		gst_datensatz.st_wkz.nockenschaltwerk_bestueckachse.arr_nocken[NO_BW_BANDFAENGER_EINFAHREN].b_camvalid := FALSE;
		gst_datensatz.st_wkz.nockenschaltwerk_bestueckachse.arr_nocken[NO_BW_BANDFAENGER_AUSFAHREN].b_camvalid := FALSE;
		gst_datensatz.st_wkz.nockenschaltwerk_bestueckachse.arr_nocken[NO_BW_BANDKLEMMEN_EINFAHREN].b_camvalid := FALSE;
		gst_datensatz.st_wkz.nockenschaltwerk_bestueckachse.arr_nocken[NO_BW_BANDKLEMMEN_AUSFAHREN].b_camvalid := FALSE;
		gst_datensatz.st_wkz.nockenschaltwerk_bestueckachse.arr_nocken[NO_UW_BANDFAENGER_EINFAHREN].b_camvalid := FALSE;
		gst_datensatz.st_wkz.nockenschaltwerk_bestueckachse.arr_nocken[NO_UW_BANDFAENGER_AUSFAHREN].b_camvalid := FALSE;
		gst_datensatz.st_wkz.nockenschaltwerk_bestueckachse.arr_nocken[NO_UW_BANDKLEMMEN_EINFAHREN].b_camvalid := FALSE;
		gst_datensatz.st_wkz.nockenschaltwerk_bestueckachse.arr_nocken[NO_UW_BANDKLEMMEN_AUSFAHREN].b_camvalid := FALSE;

		gst_datensatz.st_wkz.nockenschaltwerk_bestueckachse.arr_nocken[NO_PNEUMATIKBANDEINZUG_GLS].b_camvalid := FALSE;
		gst_datensatz.st_wkz.nockenschaltwerk_bestueckachse.arr_nocken[NO_UW_BESTUECKSCHIEBER_ON].b_camvalid := FALSE;
		gst_datensatz.st_wkz.nockenschaltwerk_bestueckachse.arr_nocken[NO_UW_BESTUECKSCHIEBER_OFF].b_camvalid := FALSE;
		gst_datensatz.st_wkz.nockenschaltwerk_bestueckachse.arr_nocken[SP_UW_BESTUECKSCHIEBER_ON].b_camvalid := FALSE;
		gst_datensatz.st_wkz.nockenschaltwerk_bestueckachse.arr_nocken[SP_UW_BESTUECKSCHIEBER_OFF].b_camvalid := FALSE;


		zyl_bandfaenger.fb.b_no_gesteuert_im_norm_betrieb := TRUE;
		zyl_bandklemmen.fb.b_no_gesteuert_im_norm_betrieb := TRUE;

		zyl_bandfaenger.fb.b_no_gesteuert_im_norm_betrieb := TRUE;
		zyl_bandklemmen.fb.b_no_gesteuert_im_norm_betrieb := TRUE;

END_CASE;
END_ACTION
ACTION subr_ST_Bandeinzugsnocken_ein:
CASE gst_datensatz.st_wkz.i16_typ_bandeinzug OF
	 STANDARD_2FACH_V2:

		(* Bandeinzug: Standard_2fach_V2 *)
		gst_datensatz.st_wkz.nockenschaltwerk_bestueckachse.arr_nocken[NO_BW_BANDFAENGER_LI_EINFAHREN].b_camvalid := TRUE;
		gst_datensatz.st_wkz.nockenschaltwerk_bestueckachse.arr_nocken[NO_BW_BANDFAENGER_LI_AUSFAHREN].b_camvalid := TRUE;
		gst_datensatz.st_wkz.nockenschaltwerk_bestueckachse.arr_nocken[NO_BW_BANDKLEMMEN_LI_EINFAHREN].b_camvalid := TRUE;
		gst_datensatz.st_wkz.nockenschaltwerk_bestueckachse.arr_nocken[NO_BW_BANDKLEMMEN_LI_AUSFAHREN].b_camvalid := TRUE;
		gst_datensatz.st_wkz.nockenschaltwerk_bestueckachse.arr_nocken[NO_UW_BANDFAENGER_LI_EINFAHREN].b_camvalid := TRUE;
		gst_datensatz.st_wkz.nockenschaltwerk_bestueckachse.arr_nocken[NO_UW_BANDFAENGER_LI_AUSFAHREN].b_camvalid := TRUE;
		gst_datensatz.st_wkz.nockenschaltwerk_bestueckachse.arr_nocken[NO_UW_BANDKLEMMEN_LI_EINFAHREN].b_camvalid := TRUE;
		gst_datensatz.st_wkz.nockenschaltwerk_bestueckachse.arr_nocken[NO_UW_BANDKLEMMEN_LI_AUSFAHREN].b_camvalid := TRUE;
		gst_datensatz.st_wkz.nockenschaltwerk_bestueckachse.arr_nocken[NO_BW_BANDFAENGER_RE_EINFAHREN].b_camvalid := TRUE;
		gst_datensatz.st_wkz.nockenschaltwerk_bestueckachse.arr_nocken[NO_BW_BANDFAENGER_RE_AUSFAHREN].b_camvalid := TRUE;
		gst_datensatz.st_wkz.nockenschaltwerk_bestueckachse.arr_nocken[NO_BW_BANDKLEMMEN_RE_EINFAHREN].b_camvalid := TRUE;
		gst_datensatz.st_wkz.nockenschaltwerk_bestueckachse.arr_nocken[NO_BW_BANDKLEMMEN_RE_AUSFAHREN].b_camvalid := TRUE;
		gst_datensatz.st_wkz.nockenschaltwerk_bestueckachse.arr_nocken[NO_UW_BANDFAENGER_RE_EINFAHREN].b_camvalid := TRUE;
		gst_datensatz.st_wkz.nockenschaltwerk_bestueckachse.arr_nocken[NO_UW_BANDFAENGER_RE_AUSFAHREN].b_camvalid := TRUE;
		gst_datensatz.st_wkz.nockenschaltwerk_bestueckachse.arr_nocken[NO_UW_BANDKLEMMEN_RE_EINFAHREN].b_camvalid := TRUE;
		gst_datensatz.st_wkz.nockenschaltwerk_bestueckachse.arr_nocken[NO_UW_BANDKLEMMEN_RE_AUSFAHREN].b_camvalid := TRUE;
		(* Bandeinzug: Standard_2fach_V2 *)
		gst_datensatz.st_wkz.nockenschaltwerk_bestueckachse.arr_nocken[NO_BW_BANDFAENGER_LI_BAEZV2_EINFAHREN].b_camvalid := TRUE;
		gst_datensatz.st_wkz.nockenschaltwerk_bestueckachse.arr_nocken[NO_BW_BANDFAENGER_LI_BAEZV2_AUSFAHREN].b_camvalid := TRUE;
		gst_datensatz.st_wkz.nockenschaltwerk_bestueckachse.arr_nocken[NO_BW_BANDKLEMMEN_LI_BAEZV2_EINFAHREN].b_camvalid := TRUE;
		gst_datensatz.st_wkz.nockenschaltwerk_bestueckachse.arr_nocken[NO_BW_BANDKLEMMEN_LI_BAEZV2_AUSFAHREN].b_camvalid := TRUE;
		gst_datensatz.st_wkz.nockenschaltwerk_bestueckachse.arr_nocken[NO_BW_BANDFAENGER_RE_BAEZV2_EINFAHREN].b_camvalid := TRUE;
		gst_datensatz.st_wkz.nockenschaltwerk_bestueckachse.arr_nocken[NO_BW_BANDFAENGER_RE_BAEZV2_AUSFAHREN].b_camvalid := TRUE;
		gst_datensatz.st_wkz.nockenschaltwerk_bestueckachse.arr_nocken[NO_BW_BANDKLEMMEN_RE_BAEZV2_EINFAHREN].b_camvalid := TRUE;
		gst_datensatz.st_wkz.nockenschaltwerk_bestueckachse.arr_nocken[NO_BW_BANDKLEMMEN_RE_BAEZV2_AUSFAHREN].b_camvalid := TRUE;

		zyl_bandfaenger_li.fb.b_no_gesteuert_im_norm_betrieb := FALSE;
		zyl_bandklemmen_li.fb.b_no_gesteuert_im_norm_betrieb := FALSE;
		zyl_bandfaenger_re.fb.b_no_gesteuert_im_norm_betrieb := FALSE;
		zyl_bandklemmen_re.fb.b_no_gesteuert_im_norm_betrieb := FALSE;

	BANDWECHSLER_V2:
		(* Klemmbandeinzug ohne Sensoren *)
		gst_datensatz.st_wkz.nockenschaltwerk_bestueckachse.arr_nocken[NO_BW_BANDFAENGER_BAWEV2_EINFAHREN].b_camvalid := TRUE;
		gst_datensatz.st_wkz.nockenschaltwerk_bestueckachse.arr_nocken[NO_BW_BANDFAENGER_BAWEV2_AUSFAHREN].b_camvalid := TRUE;
		gst_datensatz.st_wkz.nockenschaltwerk_bestueckachse.arr_nocken[NO_BW_BANDKLEMMEN_BAWEV2_EINFAHREN].b_camvalid := TRUE;
		gst_datensatz.st_wkz.nockenschaltwerk_bestueckachse.arr_nocken[NO_BW_BANDKLEMMEN_BAWEV2_AUSFAHREN].b_camvalid := TRUE;

		gst_datensatz.st_wkz.nockenschaltwerk_bestueckachse.arr_nocken[NO_BW_BANDFAENGER_EINFAHREN].b_camvalid := TRUE;
		gst_datensatz.st_wkz.nockenschaltwerk_bestueckachse.arr_nocken[NO_BW_BANDFAENGER_AUSFAHREN].b_camvalid := TRUE;
		gst_datensatz.st_wkz.nockenschaltwerk_bestueckachse.arr_nocken[NO_BW_BANDKLEMMEN_EINFAHREN].b_camvalid := TRUE;
		gst_datensatz.st_wkz.nockenschaltwerk_bestueckachse.arr_nocken[NO_BW_BANDKLEMMEN_AUSFAHREN].b_camvalid := TRUE;
		gst_datensatz.st_wkz.nockenschaltwerk_bestueckachse.arr_nocken[NO_UW_BANDFAENGER_EINFAHREN].b_camvalid := TRUE;
		gst_datensatz.st_wkz.nockenschaltwerk_bestueckachse.arr_nocken[NO_UW_BANDFAENGER_AUSFAHREN].b_camvalid := TRUE;
		gst_datensatz.st_wkz.nockenschaltwerk_bestueckachse.arr_nocken[NO_UW_BANDKLEMMEN_EINFAHREN].b_camvalid := TRUE;
		gst_datensatz.st_wkz.nockenschaltwerk_bestueckachse.arr_nocken[NO_UW_BANDKLEMMEN_AUSFAHREN].b_camvalid := TRUE;

		gst_datensatz.st_wkz.nockenschaltwerk_bestueckachse.arr_nocken[NO_PNEUMATIKBANDEINZUG_GLS].b_camvalid := TRUE;
		gst_datensatz.st_wkz.nockenschaltwerk_bestueckachse.arr_nocken[NO_UW_BESTUECKSCHIEBER_ON].b_camvalid := b_bestueckschieber_ueberwachung_aktiv;
		gst_datensatz.st_wkz.nockenschaltwerk_bestueckachse.arr_nocken[NO_UW_BESTUECKSCHIEBER_OFF].b_camvalid := b_bestueckschieber_ueberwachung_aktiv;
		gst_datensatz.st_wkz.nockenschaltwerk_bestueckachse.arr_nocken[SP_UW_BESTUECKSCHIEBER_ON].b_camvalid := b_bestueckschieber_ueberwachung_aktiv;
		gst_datensatz.st_wkz.nockenschaltwerk_bestueckachse.arr_nocken[SP_UW_BESTUECKSCHIEBER_OFF].b_camvalid := b_bestueckschieber_ueberwachung_aktiv;

		zyl_bandfaenger.fb.b_no_gesteuert_im_norm_betrieb := TRUE;
		zyl_bandklemmen.fb.b_no_gesteuert_im_norm_betrieb := TRUE;
END_CASE;
END_ACTION
ACTION subr_ST_Bandeinzugsnocken_li_ein:
CASE gst_datensatz.st_wkz.i16_typ_bandeinzug OF
	STANDARD_2FACH_V2:

		(* Bandeinzug: Standard_2fach_V1 *)
		gst_datensatz.st_wkz.nockenschaltwerk_bestueckachse.arr_nocken[NO_BW_BANDFAENGER_LI_EINFAHREN].b_camvalid := TRUE;
		gst_datensatz.st_wkz.nockenschaltwerk_bestueckachse.arr_nocken[NO_BW_BANDFAENGER_LI_AUSFAHREN].b_camvalid := TRUE;
		gst_datensatz.st_wkz.nockenschaltwerk_bestueckachse.arr_nocken[NO_BW_BANDKLEMMEN_LI_EINFAHREN].b_camvalid := TRUE;
		gst_datensatz.st_wkz.nockenschaltwerk_bestueckachse.arr_nocken[NO_BW_BANDKLEMMEN_LI_AUSFAHREN].b_camvalid := TRUE;
		gst_datensatz.st_wkz.nockenschaltwerk_bestueckachse.arr_nocken[NO_UW_BANDFAENGER_LI_EINFAHREN].b_camvalid := TRUE;
		gst_datensatz.st_wkz.nockenschaltwerk_bestueckachse.arr_nocken[NO_UW_BANDFAENGER_LI_AUSFAHREN].b_camvalid := TRUE;
		gst_datensatz.st_wkz.nockenschaltwerk_bestueckachse.arr_nocken[NO_UW_BANDKLEMMEN_LI_EINFAHREN].b_camvalid := TRUE;
		gst_datensatz.st_wkz.nockenschaltwerk_bestueckachse.arr_nocken[NO_UW_BANDKLEMMEN_LI_AUSFAHREN].b_camvalid := TRUE;
		(* Bandeinzug: Standard_2fach_V2 *)
		gst_datensatz.st_wkz.nockenschaltwerk_bestueckachse.arr_nocken[NO_BW_BANDFAENGER_LI_BAEZV2_EINFAHREN].b_camvalid := TRUE;
		gst_datensatz.st_wkz.nockenschaltwerk_bestueckachse.arr_nocken[NO_BW_BANDFAENGER_LI_BAEZV2_AUSFAHREN].b_camvalid := TRUE;
		gst_datensatz.st_wkz.nockenschaltwerk_bestueckachse.arr_nocken[NO_BW_BANDKLEMMEN_LI_BAEZV2_EINFAHREN].b_camvalid := TRUE;
		gst_datensatz.st_wkz.nockenschaltwerk_bestueckachse.arr_nocken[NO_BW_BANDKLEMMEN_LI_BAEZV2_AUSFAHREN].b_camvalid := TRUE;

		zyl_bandfaenger_li.fb.b_no_gesteuert_im_norm_betrieb := FALSE;
		zyl_bandklemmen_li.fb.b_no_gesteuert_im_norm_betrieb := FALSE;
		zyl_bandfaenger_re.fb.b_no_gesteuert_im_norm_betrieb := FALSE;
		zyl_bandklemmen_re.fb.b_no_gesteuert_im_norm_betrieb := FALSE;

END_CASE;
END_ACTION
ACTION subr_ST_Bandeinzugsnocken_re_ein:
CASE gst_datensatz.st_wkz.i16_typ_bandeinzug OF
	STANDARD_2FACH_V2:

		(* Bandeinzug: Standard_2fach_V1 *)
		gst_datensatz.st_wkz.nockenschaltwerk_bestueckachse.arr_nocken[NO_BW_BANDFAENGER_RE_EINFAHREN].b_camvalid := TRUE;
		gst_datensatz.st_wkz.nockenschaltwerk_bestueckachse.arr_nocken[NO_BW_BANDFAENGER_RE_AUSFAHREN].b_camvalid := TRUE;
		gst_datensatz.st_wkz.nockenschaltwerk_bestueckachse.arr_nocken[NO_BW_BANDKLEMMEN_RE_EINFAHREN].b_camvalid := TRUE;
		gst_datensatz.st_wkz.nockenschaltwerk_bestueckachse.arr_nocken[NO_BW_BANDKLEMMEN_RE_AUSFAHREN].b_camvalid := TRUE;
		gst_datensatz.st_wkz.nockenschaltwerk_bestueckachse.arr_nocken[NO_UW_BANDFAENGER_RE_EINFAHREN].b_camvalid := TRUE;
		gst_datensatz.st_wkz.nockenschaltwerk_bestueckachse.arr_nocken[NO_UW_BANDFAENGER_RE_AUSFAHREN].b_camvalid := TRUE;
		gst_datensatz.st_wkz.nockenschaltwerk_bestueckachse.arr_nocken[NO_UW_BANDKLEMMEN_RE_EINFAHREN].b_camvalid := TRUE;
		gst_datensatz.st_wkz.nockenschaltwerk_bestueckachse.arr_nocken[NO_UW_BANDKLEMMEN_RE_AUSFAHREN].b_camvalid := TRUE;
		(* Bandeinzug: Standard_2fach_V2 *)
		gst_datensatz.st_wkz.nockenschaltwerk_bestueckachse.arr_nocken[NO_BW_BANDFAENGER_RE_BAEZV2_EINFAHREN].b_camvalid := TRUE;
		gst_datensatz.st_wkz.nockenschaltwerk_bestueckachse.arr_nocken[NO_BW_BANDFAENGER_RE_BAEZV2_AUSFAHREN].b_camvalid := TRUE;
		gst_datensatz.st_wkz.nockenschaltwerk_bestueckachse.arr_nocken[NO_BW_BANDKLEMMEN_RE_BAEZV2_EINFAHREN].b_camvalid := TRUE;
		gst_datensatz.st_wkz.nockenschaltwerk_bestueckachse.arr_nocken[NO_BW_BANDKLEMMEN_RE_BAEZV2_AUSFAHREN].b_camvalid := TRUE;
		
		zyl_bandfaenger_li.fb.b_no_gesteuert_im_norm_betrieb := FALSE;
		zyl_bandklemmen_li.fb.b_no_gesteuert_im_norm_betrieb := FALSE;
		zyl_bandfaenger_re.fb.b_no_gesteuert_im_norm_betrieb := FALSE;
		zyl_bandklemmen_re.fb.b_no_gesteuert_im_norm_betrieb := FALSE;

END_CASE;
END_ACTION
ACTION subr_ST_Cam_B_Achse:
(* B-Achse *)
fb_axis_b_achse.st_camscaling_data.SlaveScaling :=
	F_Servobandeinzug_Strecke_zu_Grad(
		strecke := INT_TO_LREAL(gst_datensatz.st_bestueckprogramm.i16_b[i16_bestueckposzaehler])
			* gst_datensatz.st_band.r_raster);

IF b_achse.Status.CamScalingPending THEN
	st_sm.b_skalierung_noch_aktiv := TRUE;
	fb_state_entry.i16_next_step := FEHLER;
ELSE
	IF b_achse.NcToPlc.CoupleState = 0 THEN
		st_drive_cmd_b_achse.enu_cmd := CAM_IN_SLAVE;
	ELSE
		st_drive_cmd_b_achse.enu_cmd := CAM_SCALEING_SLAVE;
	END_IF
END_IF
END_ACTION
ACTION subr_ST_Cam_Bestueck_Maschine:
CASE gst_datensatz.st_md.i16_typ_zelle OF
	KEINE_ZELLE:
		;
	BESTUECKZELLE_1700, BESTUECKZELLE_1720:
		subr_ST_Cam_Bestueckachse();

	RASTERFOLIE:
		;
END_CASE
END_ACTION
ACTION subr_ST_Cam_Bestueckachse:
(* Bestueckachse *)
IF gst_datensatz.st_bestueckprogramm.i16_b[i16_bestueckposzaehler] <= 0 THEN
	i16_bestueckachse_cam_table_id := 6;	(* 0-Scalierung *)
	subr_ST_Bandeinzugsnocken_aus();
ELSE
	i16_bestueckachse_cam_table_id := 5;	(* 1-Scalierung *)
	subr_ST_Bandeinzugsnocken_ein();
END_IF

IF i16_bestueckachse_cam_table_id <> i16_bestueckachse_cam_table_id_alt THEN
	fb_axis_bestueckachse.mc_activation_mode_camin:= MC_CAMACTIVATION_ATMASTERCAMPOS;
	fb_axis_bestueckachse.lr_activation_position_camin := gst_datensatz.st_md.st_md_bestueckachse.lr_startposition;
	st_drive_cmd_bestueckachse.enu_cmd := CAM_IN_SLAVE;
	i16_bestueckachse_cam_table_id_alt := i16_bestueckachse_cam_table_id;
END_IF
END_ACTION
ACTION subr_ST_Cam_Y_Achse:
(* Y-Achse *)
IF i16_bestueckposzaehler = 0 THEN
	lr_ErsteBestueckposY := gst_datensatz.st_isk.lr_pos_y_0 +
						gst_datensatz.st_wkz.lr_offset_y_pos_0 +
						gst_datensatz.st_wt.lr_offset_y_pos_0 +
						gst_datensatz.st_md.lr_offset_y_pos_0 +
						gst_datensatz.st_bestueckprogramm.lr_y[0];
	fb_axis_y_achse.st_camscaling_data.SlaveScaling := fb_berechnung_override_achse.lr_skalierung_slave_achse2 := lr_ErsteBestueckposY - y_achse.NcToPlc.ActPos;
	(* Falls die Positionierung Probleme macht, könnte man auch so rechnen *)
	(*fb_axis_y_achse.st_camscaling_data.SlaveScaling := fb_berechnung_override_achse.lr_skalierung_slave_achse2 := lr_ErsteBestueckposY - gst_datensatz.st_wkz.r_wkz_einfahrpos_y;*)
ELSIF i16_bestueckposzaehler > 0 AND i16_bestueckposzaehler < gst_datensatz.st_bestueckprogramm.i32_anzahl THEN
	fb_axis_y_achse.st_camscaling_data.SlaveScaling := fb_berechnung_override_achse.lr_skalierung_slave_achse2 := gst_datensatz.st_bestueckprogramm.lr_y[i16_bestueckposzaehler] - gst_datensatz.st_bestueckprogramm.lr_y[i16_bestueckposzaehler - 1];
ELSE
	fb_axis_y_achse.st_camscaling_data.SlaveScaling := fb_berechnung_override_achse.lr_skalierung_slave_achse2 := 0.0;
END_IF
IF y_achse.Status.CamScalingPending THEN
	st_sm.b_skalierung_noch_aktiv := TRUE;
	fb_state_entry.i16_next_step := FEHLER;
ELSE
	IF y_achse.NcToPlc.CoupleState = 0 THEN
		st_drive_cmd_y_achse.enu_cmd := CAM_IN_SLAVE;
	ELSE
		st_drive_cmd_y_achse.enu_cmd := CAM_SCALEING_SLAVE;
	END_IF
END_IF
END_ACTION
ACTION subr_ST_Cam_Z_Achse:
(* Z-Achse *)
IF i16_bestueckposzaehler > 0 AND i16_bestueckposzaehler < gst_datensatz.st_bestueckprogramm.i32_anzahl THEN
	fb_axis_z_achse.st_camscaling_data.SlaveScaling := fb_berechnung_override_achse.lr_skalierung_slave_achse1 := gst_datensatz.st_bestueckprogramm.lr_z[i16_bestueckposzaehler] - gst_datensatz.st_bestueckprogramm.lr_z[i16_bestueckposzaehler - 1];
ELSE
	fb_axis_z_achse.st_camscaling_data.SlaveScaling := fb_berechnung_override_achse.lr_skalierung_slave_achse1 := 0.0;
END_IF
IF z_achse.Status.CamScalingPending THEN
	st_sm.b_skalierung_noch_aktiv := TRUE;
	fb_state_entry.i16_next_step := FEHLER;
ELSE
	IF z_achse.NcToPlc.CoupleState = 0 THEN
		st_drive_cmd_z_achse.enu_cmd := CAM_IN_SLAVE;
	ELSE
		st_drive_cmd_z_achse.enu_cmd := CAM_SCALEING_SLAVE;
	END_IF
END_IF
END_ACTION
ACTION subr_ST_EinzugLueften:
(* SP_SERVOBANDEINZUG_LUEFTEN niemals vorsteuern *)
gst_datensatz.st_wkz.nockenschaltwerk_bestueckachse.arr_nocken[SP_SERVOBANDEINZUG_LUEFTEN].t_vorsteuerzeit := t#0ms;

fb_r_trig_bandeinzug_lueften(CLK:= nockenschaltwerk_bestueckachse.fb.arr_spur[SP_SERVOBANDEINZUG_LUEFTEN], Q=> );
fb_f_trig_bandeinzug_lueften(CLK:= nockenschaltwerk_bestueckachse.fb.arr_spur[SP_SERVOBANDEINZUG_LUEFTEN], Q=> );

(* Abschalten, falls die Schrittkette beim Lüften aus irgendwelchen Gründen hängen bleibt *)
IF fb_r_trig_bandeinzug_lueften.Q AND
	i16_step_lueften > 0 THEN
		sm_fehler_achse_lueften := TRUE;
		fb_state_entry.i16_next_step := FEHLER;
END_IF


(* Schrittkette zum Einzug in Regelung setzen mit Positionsangleich  *)
CASE i16_step_lueften OF
(*=======================================================*)
	0:	(* CAM Out bei R Trig Lueftnocke *)

		(*-----------------------Weiterschaltbedingungen----------------------------*)
		IF fb_r_trig_bandeinzug_lueften.Q AND
			bestueckachse.NcToPlc.CoupleState <> 0 AND
			((NOT b_einfaedeln_aktiv_servo AND
			(* Bei einer Umfahrung soll Servo nicht lüften, weil die Fänger des WKZ das Band nicht halten *)
			gst_datensatz.st_bestueckprogramm.i16_b[i16_bestueckposzaehler] >= 1 ) OR
			(b_einfaedeln_aktiv_servo AND
			i16_einfaedelzaehler >= gst_datensatz.st_wkz.i16_einfaedelhub_lueften)) THEN		(* Nach x Einfädelhüben ist Band sicher im WKZ, dann darf Servobaneinzug wieder entlüften *)
			st_drive_cmd_b_achse.enu_cmd := CAM_OUT_SLAVE;
			i16_step_lueften := 10;
		END_IF

(*=======================================================*)
	10:

		(*-----------------------Weiterschaltbedingungen----------------------------*)
		IF st_drive_cmd_b_achse.enu_cmd = NO_COMMAND THEN
			ST_Servobandeinzug.i_Stromlimit := ST_Servobandeinzug.i16_lueft_torque;
			i16_step_lueften := 20;
		END_IF

(*=======================================================*)
	20: (* HOME Servobandeinzug bei F Trig Lueftnocke *)

		(*-----------------------Weiterschaltbedingungen----------------------------*)
		IF fb_f_trig_bandeinzug_lueften.Q THEN
			axis_bandeinzug_achse.st_ctrl.in.b_home := TRUE;
			i16_step_lueften := 30;
		END_IF

(*=======================================================*)
	30:

		(*-----------------------Weiterschaltbedingungen----------------------------*)
		IF axis_bandeinzug_achse.st_ctrl.out.b_fertig_2 THEN
			axis_bandeinzug_achse.st_ctrl.in.b_home := FALSE;
			i16_step_lueften := 0;
		END_IF

END_CASE
END_ACTION
ACTION subr_ST_PosUW_Bestueckachse:
(* Wenn die Betückachse von der Virtuellen Achse entkoppelt wird, muss dauerhaft der OT Sensor belegt sein.
Überwachung, ob das Auskoppeln rechtzeitig gemacht wird. Ab 300 Hub gibt es Probleme *)
IF i16_bestueckachse_cam_table_id = 6 AND NOT ST_Bestueckachse.e_referenz_sensor THEN
	sm_fehler_positionierung_bestueckachse := TRUE;
	fb_state_entry.i16_next_step := FEHLER;
END_IF
END_ACTION
ACTION subr_ST_PosUW_YZ_Achse:
(* Y *)
(* Kontrolle der Skalierungsposition der Achse nach dem Setzen eines Pins *)
IF ABS(y_achse.NcToPlc.ActPos - (lr_merker_y_pos + gst_datensatz.st_bestueckprogramm.lr_y[i16_bestueckposzaehler])) > 0.1THEN
	sm_fehler_bestueckposition_y := TRUE;
	fb_state_entry.i16_next_step := FEHLER;
END_IF

(* Überwachung auf Kommando abgeschlossen. Zusätzliche Kontrolle auf Ausführung des Skalierungskommandos *)
IF st_drive_cmd_y_achse.enu_cmd <> NO_COMMAND THEN
	st_sm.b_ende_camming_nocke := TRUE;
	fb_state_entry.i16_next_step := FEHLER;
END_IF

(* Z *)
(* Kontrolle der Skalierungsposition der Achse nach dem Setzen eines Pins *)
IF ABS(z_achse.NcToPlc.ActPos - (lr_merker_z_pos + gst_datensatz.st_bestueckprogramm.lr_z[i16_bestueckposzaehler])) > 0.2THEN
	sm_fehler_bestueckposition_z := TRUE;
	fb_state_entry.i16_next_step := FEHLER;
END_IF

(* Überwachung auf Kommando abgeschlossen. Zusätzliche Kontrolle auf Ausführung des Skalierungskommandos *)
IF st_drive_cmd_z_achse.enu_cmd <> NO_COMMAND THEN
	st_sm.b_ende_camming_nocke := TRUE;
	fb_state_entry.i16_next_step := FEHLER;
END_IF

(* Pythagoras YZ *)
(*	tv + gg: 10.08.2021
	Wir müssen nicht nur jede Achse einzeln überwachen, sondern beide Achsen zusammen überwachen.
	Bsp. 74pol 2-Fach WT: Es gibt hier Sprünge die nur 0.04 in Y Verschoben, welche dann die 
	Überwachung in Y-Achse ausgelöst hat, obwohl alles funktionert hat. Z Pos ist um 5 mm verschoben*)

(* Kontrolle, ob die Achsen gegenüber dem letzten Bestückhub weiter gefahren ist *)
lr_merker_y_pos_neu := y_achse.NcToPlc.ActPos;
lr_merker_z_pos_neu := z_achse.NcToPlc.ActPos;

lr_abstand_yz := SQRT(	EXPT(lr_merker_y_pos_alt - lr_merker_y_pos_neu, 2) +
						EXPT(lr_merker_z_pos_alt - lr_merker_z_pos_neu, 2));

IF 	(fb_axis_y_achse.st_camscaling_data.SlaveScaling <> 0 OR
	fb_axis_z_achse.st_camscaling_data.SlaveScaling <> 0) AND
	lr_abstand_yz < 0.05
THEN
	sm_fehler_positionierung_y := TRUE;
	sm_fehler_positionierung_z := TRUE;
	fb_state_entry.i16_next_step := FEHLER;
END_IF

lr_merker_y_pos_alt := lr_merker_y_pos_neu;
lr_merker_z_pos_alt := lr_merker_z_pos_neu;
END_ACTION
ACTION subr_ST_PosUW_Z_Achse:
(* Kontrolle der Skalierungsposition der Achse nach dem Setzen eines Pins *)
IF ABS(z_achse.NcToPlc.ActPos - (lr_merker_z_pos + gst_datensatz.st_bestueckprogramm.lr_z[i16_bestueckposzaehler])) > 0.2THEN
	sm_fehler_bestueckposition_z := TRUE;
	fb_state_entry.i16_next_step := FEHLER;
END_IF

(* Überwachung auf Kommando abgeschlossen. Zusätzliche Kontrolle auf Ausführung des Skalierungskommandos *)
IF st_drive_cmd_z_achse.enu_cmd <> NO_COMMAND THEN
	st_sm.b_ende_camming_nocke := TRUE;
	fb_state_entry.i16_next_step := FEHLER;
END_IF

(* Kontrolle, ob die Achse gegenüber dem letzten Bestückhub weiter gefahren ist *)
lr_merker_z_pos_neu := z_achse.NcToPlc.ActPos;
IF fb_axis_z_achse.st_camscaling_data.SlaveScaling <> 0 THEN
	IF ABS(lr_merker_z_pos_alt - lr_merker_z_pos_neu) > 0.05 THEN
		lr_merker_z_pos_alt := lr_merker_z_pos_neu;
	ELSE
		sm_fehler_positionierung_z := TRUE;
		fb_state_entry.i16_next_step := FEHLER;
	END_IF
END_IF
END_ACTION

(* POU EPT Lib/Funktionsbausteine/ST_BerechnungOverride, ST *)
FUNCTION_BLOCK ST_BerechnungOverride
VAR_INPUT
	i16_betriebsart				: enum_betriebsarten;
	lr_skalierung_slave_achse1		: LREAL;
	lr_skalierung_slave_achse2		: LREAL;
	lr_override_vorgabe			: LREAL;
	lr_faktor						: LREAL;

	lr_FaktorHub				: LREAL;
	lr_HubAuto					: LREAL;
END_VAR
VAR_OUTPUT
	lr_override					: LREAL := 0.0;
END_VAR
VAR
	lr_offset						: LREAL := 100.0;
	tmp_lr_override_slave1		: LREAL := 0.0;
	tmp_lr_override_slave2		: LREAL := 0.0;

	lr_ProzentDerRichtdrehzahl	: LREAL;
	lr_Reduzierung				: LREAL;
END_VAR
(* Funktion zur Berechnung des Override der  Masterachse: y = - faktor * x^2 + offset *)
(* Die Funktion besteht aus einer auf dem Kopf stehenden Parabel, welche um den faktor nach oben verschoben ist *)
(* Aufpassen bei den Nullstellen der Funktion, wenn faktor und offset verändert werden *)

(* Die Anpassung der maximalen Mastergeschwindigkeit an die Verfahrlänge des Slaves wird hier einfach über eine empirisch ermittelte Funktion realisiert *)
(* Eine verbesserte Anpassung stellt die Berechnung der maximalen Mastergeschwindigkeit (ST_MFMaxMasterVelo) im CamEditor dar. *)

tmp_lr_override_slave1 := - lr_faktor * (lr_skalierung_slave_achse1 * lr_skalierung_slave_achse1)  + lr_offset;
tmp_lr_override_slave2 := - lr_faktor * (lr_skalierung_slave_achse2 * lr_skalierung_slave_achse2)  + lr_offset;

IF tmp_lr_override_slave1 < 0.0 THEN
	 tmp_lr_override_slave1 := 0.0;
ELSIF tmp_lr_override_slave1 >= 100.0 THEN
	 tmp_lr_override_slave1 := 100.0;
END_IF
IF tmp_lr_override_slave2 < 0.0 THEN
	 tmp_lr_override_slave2 := 0.0;
ELSIF tmp_lr_override_slave2 >= 100.0 THEN
	 tmp_lr_override_slave2 := 100.0;
END_IF

IF i16_betriebsart = AUTO THEN
	(* Nur wenn der mit der Funktion berechnete Override kleiner ist, als die Vorgabe, dann wird der Funktionswert übernommen *)
	IF 	tmp_lr_override_slave1 < lr_override_vorgabe OR
		tmp_lr_override_slave2 < lr_override_vorgabe THEN

		IF tmp_lr_override_slave1 <= tmp_lr_override_slave2 THEN
			lr_override := tmp_lr_override_slave1;
		ELSIF tmp_lr_override_slave2 < tmp_lr_override_slave1 THEN
			lr_override := tmp_lr_override_slave2;
		ELSE
			lr_override := lr_override_vorgabe;
		END_IF

	ELSE
		lr_override := lr_override_vorgabe;
	END_IF
ELSE
	lr_override := lr_override_vorgabe;
END_IF


(*neue Berechnung==========================================================================*)
(*Reduzierung abhängig von der Nenndrehzahl*)
lr_ProzentDerRichtdrehzahl:=(lr_HubAuto *100)/250;
IF	lr_HubAuto >250 AND
	lr_override_vorgabe > lr_override THEN
	lr_override := 100-((lr_override_vorgabe - lr_override) * (lr_ProzentDerRichtdrehzahl /100)) ;
END_IF

(*nur Reduzieren wenn das Ergebniss kleiner ist als bei der Reduzierung durch die Pin Anzahl*)
lr_Reduzierung:= (lr_override_vorgabe - lr_override)/100;
IF	(1 - lr_Reduzierung) < lr_FaktorHub THEN
	lr_override := lr_override;
ELSE
	lr_override:= 100 * lr_FaktorHub;
END_IF

IF	lr_override > lr_override_vorgabe OR
	lr_override < 0 THEN
	lr_override:= lr_override_vorgabe;
END_IF

(*Beim Einfädeln wird der Override vom Bausstein ST_TippTasten einfach durchgeschleust*)
IF	ST_TippTasten.b_einfaedeln_aktiv OR
	ST_TippTasten.b_initialisierungsphase THEN
	lr_override := lr_override_vorgabe;
END_IF

(*bei Prüfteilen Override fest auf 30% *)
IF	lr_override_vorgabe > 30 AND
	(FIND( gst_datensatz.st_md.s_aktuelle_artikelnummer,'ruef') <> 0 OR FIND( gst_datensatz.st_md.s_aktuelle_artikelnummer,'erth') <> 0)THEN
	lr_override := 30;
END_IF
END_FUNCTION_BLOCK

(* POU Gemeinsamkeiten17xx/Achsen/ST_Servobandeinzug, ST *)
PROGRAM ST_Servobandeinzug
VAR_INPUT
	st_config_achse						: struct_ecd_config;
	st_ctrl_in								: struct_ctrl_in;
	e_steuerung_ein						: BOOL;
	e_ba_mit_bedingungen				: BOOL;
	e_tuere_vorne_offen					: BOOL;
	e_tuere_hinten_offen					: BOOL;
	i_Stromlimit							: INT;		(* Werte zwischen 0 und 1000 möglich*)
END_VAR
VAR_IN_OUT
	st_visu								: struct_ecd_visu;
END_VAR
VAR_OUTPUT
	st_ctrl_out							: struct_ctrl_out;
END_VAR
VAR
	st_sm						 		: struct_ecd_meldungen;
	st_drive_cmd							: struct_ecd_cmd;
	fb_ton_wz							: TON;
	fb_ton_quitt							: TON;
	fb_r_trig_taste_plus					: R_TRIG;
	fb_r_trig_taste_minus					: R_TRIG;
	fb_r_trig_bremse						: R_TRIG;
	fb_r_trig_tippen						: R_TRIG;
	fb_r_trig_hand_dialog					: R_TRIG;
	fb_axis								: ST_AxisJobCtrl_Motion;
	fb_state_entry							: ST_StateEntry;
	fb_ton_uez							: TON;
	b_ibn_start							: BOOL := FALSE;
	fb_r_trig_ibn_start						: R_TRIG;
	fb_ton_ibn_start						: TON;
	fb_ton_wz_rueckzug					: TON;
	fb_tof_gls_ref							: TOF;
	fb_r_trig_gls_ref						: R_TRIG;
	fb_ton_wz_disable						: TON;
	fb_ton_wz_param						: TON;
	i									: UINT := 0;
	fb_r_trig_limit_sensor_positiv			: R_TRIG;
	fb_r_trig_limit_sensor_negativ			: R_TRIG;
	fb_r_trig_achse_lueften					: R_TRIG;
	b_referenzieren						: BOOL := FALSE;

	b_hand_dialog_aktiv					: BOOL := FALSE;
	st_geschwindigkeiten					: struct_ecd_geschwindigkeiten;
	i_zaehler_steigende_flanke				: INT;	(* Zähler für Bandvorschubkontrolle Gabellichtschranke *)
	i_zaehler_fallende_flanke				: INT;	(* Zähler für Bandvorschubkontrolle Gabellichtschranke *)
	fb_r_trig_vorschubkontrolle				: R_TRIG;
	fb_f_trig_vorschubkontrolle				: F_TRIG;
	fb_r_trig_nocke_einzug					: R_TRIG;
	fb_f_trig_nocke_einzug					: F_TRIG;
	i16_max_torque						: INT := 1000;
	i16_lueft_torque						: INT := 2;	(* sehr klein, damit sich Band ausrichten kann und Servo nicht dagegen arbeitet *)
	i16_man_einfaedel_torque				: INT := 30;
	i16_auto_einfaedel_torque				: INT := 150;
	i16_einfaedel_torque					: INT := 20;
	i16_block_torque						: INT := 40;
	lr_rueckzugposition					: LREAL := 0.5;
	b_merker_bremse						: BOOL := FALSE;
	b_merker_bremse_auf_zu				: BOOL := FALSE;
	r_raster_alt							: REAL := 0.0;
	i16_raster_nc_parameter				: INT := 0;
	b_merker_lueften						: BOOL := FALSE;
	b_merker_regeln						: BOOL := FALSE;

	err_id								: DWORD := 0;

	mc_set_cam_online_change_mode		: MC_SetCamOnlineChangeMode;

	lr_posmerker_an_faenger				: LREAL := 0;

	sm_bandrueckzug						: BOOL := FALSE;
	sm_bandreferenzieren					: BOOL := FALSE;
	sm_fehler_bandvorschub				: BOOL := FALSE;
	sm_fehler_raster						: BOOL := FALSE;
	sm_fehler_bandeinfaedeln				: BOOL := FALSE;
	sm_fahren_auf_gls					: BOOL := FALSE;
	sm_band_rausgezogen				: BOOL := FALSE;
	sm_band_nicht_in_lichtschranke			: BOOL := FALSE;

	e_limit_sensor_positive				AT %I* : BOOL;
	e_limit_sensor_negative				AT %I* : BOOL;
	e_gls_bandreferenzieren				AT %I* : BOOL;	(* Sensor dient auch als Vorschubkontrolle *)
	i16_torque							AT %I* : INT;
	i16_vorgabe_stromlimit					AT %Q* : INT;

	i16_debug 							: INT;

	(* Lueften *)
	fb_r_trig_bandeinzug_lueften			: R_TRIG;

	lr_merker_pos_vor_lueften				: LREAL := 0.0;
	lr_merker_pos_nach_lueften			: LREAL := 0.0;
	lr_merker_pos_diff_lueften				: LREAL := 0.0;

	lr_startpos							: LREAL := 0;

END_VAR

VAR CONSTANT
	lr_konst_strecke_ls_bandeinzug			: LREAL := 70;
	lr_max_strecke_gls_wkz				: LREAL := 110;
END_VAR
(* Zeiten *)
fb_ton_wz(IN:= , PT:= , Q=>  , ET=> );
fb_ton_uez(IN:= , PT:= , Q=>  , ET=> );
fb_ton_wz_rueckzug(IN:= , PT:= t#300ms, Q=> , ET=> );
fb_tof_gls_ref(IN:= e_gls_bandreferenzieren, PT:= t#150ms, Q=>  , ET=> );
fb_ton_wz_disable(IN:= , PT:= t#500ms, Q=> , ET=> );
fb_ton_wz_param(IN:= , PT:= t#500ms, Q=> , ET=> );
fb_ton_quitt(IN:= , PT:= t#100ms, Q=> , ET=> );


(* Flanken *)
fb_r_trig_limit_sensor_positiv(CLK:= st_config_achse.b_limitsensor_positiv_vorhanden AND NOT e_limit_sensor_positive, Q=> );
fb_r_trig_limit_sensor_negativ(CLK:= st_config_achse.b_limitsensor_negativ_vorhanden AND NOT e_limit_sensor_negative, Q=> );
fb_r_trig_taste_plus(CLK:= ST_Euchner_Handbedienpult.b_Taste_Plus, Q=> );
fb_r_trig_taste_minus(CLK:= ST_Euchner_Handbedienpult.b_Taste_Minus, Q=> );
fb_r_trig_bremse(CLK:= visu_hinten.out.ST_Servobandeinzug.b_taste_bremse, Q=> );
fb_r_trig_tippen(CLK:= visu_hinten.out.ST_Servobandeinzug.b_taste_tippen, Q=> );
fb_r_trig_gls_ref(CLK:= e_gls_bandreferenzieren, Q=> );
fb_r_trig_vorschubkontrolle(CLK:= e_gls_bandreferenzieren, Q=> );
fb_f_trig_vorschubkontrolle(CLK:= e_gls_bandreferenzieren, Q=> );

fb_r_trig_hand_dialog(CLK:= b_hand_dialog_aktiv, Q=> );

fb_f_trig_nocke_einzug(CLK:= nockenschaltwerk_bestueckachse.fb.arr_spur[SP_SERVOBANDEINZUG_GLS], Q=> );
fb_r_trig_nocke_einzug(CLK:= nockenschaltwerk_bestueckachse.fb.arr_spur[SP_SERVOBANDEINZUG_GLS], Q=> );

(* Inbetriebnahme *)
fb_r_trig_ibn_start (CLK:= b_ibn_start , Q=> );
fb_ton_ibn_start (IN:= , PT:= t#1s, Q=> , ET=> );

i16_debug := fb_state_entry.i16_step;

IF fb_r_trig_ibn_start .Q THEN
	fb_ton_ibn_start .IN := TRUE;
ELSE
	IF fb_ton_ibn_start .Q THEN
		b_ibn_start  := FALSE;
	 	fb_ton_ibn_start .IN := FALSE;
	END_IF
END_IF

(* Vorgabewert an Regler übergeben*)
i16_vorgabe_stromlimit := i_Stromlimit;

(* Achse steuern *)
IF fb_state_entry.i16_step >= 500 AND fb_state_entry.i16_step < 700 THEN
	fb_axis.lr_override_vorgabe := 3.0;
ELSIF fb_state_entry.i16_step >= 700 AND fb_state_entry.i16_step < 800 THEN
	fb_axis.lr_override_vorgabe := 25.0;
ELSE
	fb_axis.lr_override_vorgabe := ST_TippTasten.lr_override;
END_IF

fb_axis(
	e_referenznocken:= ,
	b_refsensor_vorhanden:= st_config_achse.b_refsensor_vorhanden,
	b_limitsensor_positiv_vorhanden:= st_config_achse.b_limitsensor_positiv_vorhanden,
	b_limitsensor_negativ_vorhanden:= st_config_achse.b_limitsensor_negativ_vorhanden,
	i16_achstyp := st_config_achse.i16_achstyp,
	st_position:= ,
	lr_override_vorgabe:= ,
	mc_richtung_modulo:= ,
	mc_richtung_velocity:= ,
	mc_referenzmodus:= ,
	mc_buffermode_axis:= ,
	ui16_soeparam_write_value:= ,
	w_idn:= ,
	i16_nc_parameter_nummer:= ,
	r_wert_nc_write_parameter:= ,
	st_vorgabe_geschwindigkeiten:= st_geschwindigkeiten,
	lr_soll_geschwindigkeit:=,
	b_bedingung_sls:= NOT e_tuere_vorne_offen OR NOT e_tuere_hinten_offen,
	st_ads_info := ,
	st_eccoe_sdo := ,
	st_masterachse:= b_achse,
	st_visu_axis:= st_visu,
	st_ecd_cmd:= st_drive_cmd,
	ui16_soeparam_read_value=> ,
	r_wert_nc_read_parameter=> );

(* Achse mit dem Euchner Handbediengerät vorwärts und rückwärts Bewegen*)
IF ST_Betriebsarten.i16_betriebsart = HAND AND fb_r_trig_hand_dialog.Q THEN
	fb_state_entry.i16_next_step := HANDRAD;
END_IF

(* Visualisierung des Bremsenzustandes am Backpanel *)
IF fb_axis.ui16_soeparam_write_value = 0 THEN
	 visu_hinten.in.b_zustand_bremse := FALSE;
ELSIF fb_axis.ui16_soeparam_write_value = 2 THEN
	 visu_hinten.in.b_zustand_bremse := TRUE;
END_IF

(* Motorbremse von Hand am Backpanel öffnen *)
IF fb_r_trig_bremse.Q THEN
	fb_ton_wz_disable.IN := FALSE;
	fb_ton_wz_param.IN := FALSE;
	b_merker_bremse := TRUE;
END_IF

IF b_merker_bremse THEN
	(* Reglerfreigabe wegnehmen/setzen und Motorbremse auf/zu *)
	IF NOT fb_ton_wz_disable.IN AND NOT fb_ton_wz_param.IN THEN
		IF b_merker_bremse_auf_zu THEN
			(* Bremse ZU *)
			st_drive_cmd.enu_cmd := POWER_ENABLE;
			fb_axis.ui16_soeparam_write_value := 0;
			b_merker_bremse_auf_zu := FALSE;
		ELSE
			(* Bremse AUF *)
			st_drive_cmd.enu_cmd := POWER_DISABLE;
			fb_axis.ui16_soeparam_write_value := 2;
			b_merker_bremse_auf_zu := TRUE;
		END_IF
		fb_ton_wz_disable.IN := TRUE;
	END_IF

	IF fb_ton_wz_disable.Q AND st_drive_cmd.enu_cmd = NO_COMMAND THEN
		fb_axis.w_idn := P_0_IDN + 96;
		st_drive_cmd.enu_cmd := SOE_WRITE_PARAM;
		fb_ton_wz_disable.IN := FALSE;
		fb_ton_wz_param.IN := TRUE;
	END_IF

	IF fb_ton_wz_param.Q AND st_drive_cmd.enu_cmd = NO_COMMAND THEN
		fb_ton_wz_param.IN := FALSE;
		b_merker_bremse := FALSE;
	END_IF
END_IF

(* Vorschubkontrolle des Bandes *)
IF fb_state_entry.i16_next_step >= BEREIT AND fb_state_entry.i16_next_step < 400 THEN
	subr_ST_Vorschubkontrolle();
END_IF

(* =======================================Toplevel========================================== *)
(* Starte Inbetriebnahme-Sequenz *)
IF st_ctrl_in.b_gehe_step_ibn THEN
	fb_state_entry.i16_next_step := INBETRIEBNAHME;
END_IF

IF (NOT e_steuerung_ein OR NOT e_ba_mit_bedingungen) AND y_achse.Status.Operational THEN
	st_drive_cmd.enu_cmd := POWER_DISABLE;
END_IF

IF fb_state_entry.i16_next_step > INIT AND fb_state_entry.i16_next_step < FEHLER THEN
	(* =====Fehler vom Achskontroller===== *)
	IF st_drive_cmd.b_job_fehler THEN
		fb_state_entry.i16_next_step := FEHLER;
	END_IF

	IF fb_state_entry.i16_next_step > 70 THEN
		(* Devicefehler *)
		IF b_achse.Status.Error THEN
			st_sm.b_achsfehler := TRUE;
			(*  Bei einem Achsfehler des Servomotors wird das Drehmoment weggeschalten, um ein Zerstören des Igelrads zu vermeiden. *)
			i_Stromlimit := i16_lueft_torque;
			fb_state_entry.i16_next_step := FEHLER;
		ELSIF b_achse.Status.DriveDeviceError THEN
			st_sm.b_devicefehler := TRUE;
			fb_state_entry.i16_next_step := FEHLER;
		END_IF
	END_IF

	IF fb_state_entry.i16_next_step < STOP THEN
		(* =====Achse wird gestoppt===== *)
		IF st_ctrl_in.b_stop THEN
			fb_state_entry.i16_next_step := STOP;
		ELSIF fb_state_entry.i16_next_step < HALT THEN
			(* =====Achse wird angehalten===== *)
			IF st_ctrl_in.b_halt THEN
				fb_state_entry.i16_next_step := HALT;
			END_IF
		END_IF
	END_IF
END_IF

(* ==================================Schrittkette================================ *)
fb_state_entry(
	i16_next_step:= ,
	i16_pos:= 1,
	s_debugtext:= ,
	E=> ,
	X=> ,
	i16_step=> ,
	i16_last_step=> );

CASE fb_state_entry.i16_step OF
(*=======================================================*)
	INIT_OBJ:
		IF st_config_achse.b_config_fertig THEN
			fb_state_entry.i16_next_step := 1;
		END_IF

(*=======================================================*)
	1:	(* Warte bis NetID´s der Slaves ausgelesen sind *)
		IF fb_state_entry.E THEN
			;
		END_IF

		(*-----------------------Weiterschaltbedingungen----------------------------*)
		IF ST_EthercatDiag.st_ctrl_out.b_fertig THEN
			fb_state_entry.i16_next_step := 2;
		END_IF

(*=======================================================*)
	2:	(* Spezifische NC-Achsparameter auslesen *)
		IF fb_state_entry.E THEN
			fb_axis.i16_nc_parameter_nummer := MaxVelocitySystem;
			st_drive_cmd.enu_cmd := READ_NC_PARAMETER;
		END_IF

		(*-----------------------Weiterschaltbedingungen----------------------------*)
		IF st_drive_cmd.enu_cmd = NO_COMMAND THEN
			st_geschwindigkeiten.lr_auto_max := fb_axis.r_wert_nc_read_parameter;
			st_geschwindigkeiten.lr_maximalgeschwindigkeit := fb_axis.r_wert_nc_read_parameter;
			st_geschwindigkeiten.lr_auto_min := 1;
			st_geschwindigkeiten.lr_jog := 50;
			fb_state_entry.i16_next_step := 3;
		END_IF

(*=======================================================*)
	3:	(* Spezifische NC-Achsparameter auslesen *)
		IF fb_state_entry.E THEN
			fb_axis.i16_nc_parameter_nummer := MaxAccelerationSystem;
			st_drive_cmd.enu_cmd := READ_NC_PARAMETER;
		END_IF

		(*-----------------------Weiterschaltbedingungen----------------------------*)
		IF st_drive_cmd.enu_cmd = NO_COMMAND THEN
			st_geschwindigkeiten.lr_beschleunigung := fb_axis.r_wert_nc_read_parameter;
			fb_state_entry.i16_next_step := 4;
		END_IF

(*=======================================================*)
	4:	(* Spezifische NC-Achsparameter auslesen *)
		IF fb_state_entry.E THEN
			fb_axis.i16_nc_parameter_nummer := MaxDecelerationSystem;
			st_drive_cmd.enu_cmd := READ_NC_PARAMETER;
		END_IF

		(*-----------------------Weiterschaltbedingungen----------------------------*)
		IF st_drive_cmd.enu_cmd = NO_COMMAND THEN
			st_geschwindigkeiten.lr_verzoegerung := fb_axis.r_wert_nc_read_parameter;
			fb_state_entry.i16_next_step := 5;
		END_IF

(*=======================================================*)
	5:	(* Spezifische NC-Achsparameter auslesen *)
		IF fb_state_entry.E THEN
			fb_axis.i16_nc_parameter_nummer := MaxJerk;
			st_drive_cmd.enu_cmd := READ_NC_PARAMETER;
		END_IF

		(*-----------------------Weiterschaltbedingungen----------------------------*)
		IF st_drive_cmd.enu_cmd = NO_COMMAND THEN
			st_geschwindigkeiten.lr_ruck := fb_axis.r_wert_nc_read_parameter;
			fb_state_entry.i16_next_step := 6;
		END_IF

(*=======================================================*)
	6:	(* Konfigurationen der Achse *)
		IF fb_state_entry.E THEN
			fb_axis.st_eccoe_sdo.s_ec_slave_net_id := ST_EthercatDiag.s_ec_slave_net_id[2];
			fb_axis.st_eccoe_sdo.ui16_slave_addr := st_config_achse.ui16_ethercat_adr;
		END_IF

		(*-----------------------Weiterschaltbedingungen----------------------------*)
		fb_state_entry.i16_next_step := FEHLER; (*in Fehler gehen damit die Achsen resetet werden. Sonst steigen die Achsen bei einem TC Restart aus*)

(*=======================================================*)
	INIT:
		IF fb_state_entry.E THEN
			fb_ton_wz.IN := FALSE;
			fb_ton_uez.IN	:= FALSE;
			fb_ton_quitt.IN := FALSE;
			fb_ton_wz_rueckzug.IN := FALSE;
			fb_tof_gls_ref.IN := FALSE;
			fb_ton_wz_disable.IN := FALSE;
			b_referenzieren := FALSE;
			sm_bandrueckzug := FALSE;
			sm_bandreferenzieren := FALSE;
			sm_fehler_bandvorschub := FALSE;
			sm_fehler_raster := FALSE;
			sm_fehler_bandeinfaedeln := FALSE;
			sm_fahren_auf_gls := FALSE;
			sm_band_rausgezogen := FALSE;
			sm_band_nicht_in_lichtschranke := FALSE;
			st_sm.b_achse_nicht_auf_startpos := FALSE;
			st_sm.b_achsfehler := FALSE;
			st_sm.b_devicefehler := FALSE;
			st_sm.b_keine_verfahrfreigabe := FALSE;
			st_sm.b_ende_skalierungs_nocke := FALSE;
			st_sm.b_ende_camming_nocke := FALSE;
			st_sm.b_skalierung_noch_aktiv := FALSE;
			st_ctrl_out.b_fehler := FALSE;
			st_ctrl_out.b_fertig := FALSE;
			st_ctrl_out.b_fertig_2 := FALSE;
			st_ctrl_out.b_bereit := FALSE;
			st_ctrl_out.b_prebereit := FALSE;
			st_ctrl_out.b_bandende := FALSE;
			st_ctrl_out.b_bremse_geoeffnet := FALSE;
			st_ctrl_out.b_bremse_geschlossen := FALSE;
			st_ctrl_out.b_servo_auf_einfaedelpos := FALSE;
			i16_max_torque := 1000;
			i16_lueft_torque := 2;	(* sehr klein, damit sich Band ausrichten kann und Servo nicht dagegen arbeitet *)
			i16_man_einfaedel_torque := 30;
			i16_auto_einfaedel_torque := 150;
			i16_einfaedel_torque := 20;
			i16_block_torque := 40;
			i_Stromlimit := i16_max_torque;
			mc_set_cam_online_change_mode.Execute := FALSE;

			fb_axis.lr_soll_geschwindigkeit := gst_datensatz.st_wkz.r_auto_bandeinzug;
		END_IF

		(*-----------------------Weiterschaltbedingungen----------------------------*)
		IF st_ctrl_in.b_preinit THEN
			fb_state_entry.i16_next_step := 20;
		END_IF

(*=======================================================*)
	20:	(* Schleppabstandsüberwachung einschalten *)
		IF fb_state_entry.E THEN
			fb_axis.r_wert_nc_write_parameter := 1;
			fb_axis.i16_nc_parameter_nummer := EnablePosLagMonitoring;
			st_drive_cmd.enu_cmd := WRITE_NC_PARAMETER;
		END_IF

		(*-----------------------Weiterschaltbedingungen----------------------------*)
		IF st_drive_cmd.enu_cmd = NO_COMMAND THEN
			fb_state_entry.i16_next_step := 25;
		END_IF

(*=======================================================*)
	25:	(* Abfrage auf geändertes Raster *)

		(*-----------------------Weiterschaltbedingungen----------------------------*)
		IF r_raster_alt = gst_datensatz.st_band.r_raster THEN
			fb_state_entry.i16_next_step := 60;
		ELSE
			fb_state_entry.i16_next_step := 30;	(* Rasterwechsel -> NC-Parameter müssen neu eingelesen werden! *)
		END_IF

(*=======================================================*)
	30:	(* Konfiguration der Achse in Abhängigkeit des Igelrades/Rasters *)
		(* Die Werte wurden in der Achs-Konfiguration des Systemmanagers für die verschiedenen Raster berechnet *)
		IF fb_state_entry.E THEN
			fb_state_entry.i16_next_step := 41;
		END_IF

(*=======================================================*)
	41:	(* Spezifische NC-Achsparameter auslesen *)
		IF fb_state_entry.E THEN
			fb_axis.i16_nc_parameter_nummer := MaxVelocitySystem;
			st_drive_cmd.enu_cmd := READ_NC_PARAMETER;
		END_IF

		(*-----------------------Weiterschaltbedingungen----------------------------*)
		IF st_drive_cmd.enu_cmd = NO_COMMAND THEN
			st_geschwindigkeiten.lr_auto_max := fb_axis.r_wert_nc_read_parameter;
			st_geschwindigkeiten.lr_maximalgeschwindigkeit := fb_axis.r_wert_nc_read_parameter;
			st_geschwindigkeiten.lr_auto_min := 1;
			st_geschwindigkeiten.lr_jog :=360;
			fb_state_entry.i16_next_step := 42;
		END_IF

(*=======================================================*)
	42:	(* Spezifische NC-Achsparameter auslesen *)
		IF fb_state_entry.E THEN
			fb_axis.i16_nc_parameter_nummer := MaxAccelerationSystem;
			st_drive_cmd.enu_cmd := READ_NC_PARAMETER;
		END_IF

		(*-----------------------Weiterschaltbedingungen----------------------------*)
		IF st_drive_cmd.enu_cmd = NO_COMMAND THEN
			st_geschwindigkeiten.lr_beschleunigung := fb_axis.r_wert_nc_read_parameter;
			fb_state_entry.i16_next_step := 43;
		END_IF

(*=======================================================*)
	43:	(* Spezifische NC-Achsparameter auslesen *)
		IF fb_state_entry.E THEN
			fb_axis.i16_nc_parameter_nummer := MaxDecelerationSystem;
			st_drive_cmd.enu_cmd := READ_NC_PARAMETER;
		END_IF

		(*-----------------------Weiterschaltbedingungen----------------------------*)
		IF st_drive_cmd.enu_cmd = NO_COMMAND THEN
			st_geschwindigkeiten.lr_verzoegerung := fb_axis.r_wert_nc_read_parameter;
			fb_state_entry.i16_next_step := 44;
		END_IF

(*=======================================================*)
	44:	(* Spezifische NC-Achsparameter auslesen *)
		IF fb_state_entry.E THEN
			fb_axis.i16_nc_parameter_nummer := MaxJerk;
			st_drive_cmd.enu_cmd := READ_NC_PARAMETER;
		END_IF

		(*-----------------------Weiterschaltbedingungen----------------------------*)
		IF st_drive_cmd.enu_cmd = NO_COMMAND THEN
			st_geschwindigkeiten.lr_ruck := fb_axis.r_wert_nc_read_parameter;
			fb_state_entry.i16_next_step := 45;
		END_IF

(*=======================================================*)
	45:	(* Bremse auf "automtisch" stellen. *)
		IF fb_state_entry.E THEN
			fb_axis.w_idn := P_0_IDN + 96;
			fb_axis.ui16_soeparam_write_value := 0;
			st_drive_cmd.enu_cmd := SOE_WRITE_PARAM;
		END_IF

		(*-----------------------Weiterschaltbedingungen----------------------------*)
		IF st_drive_cmd.enu_cmd = NO_COMMAND THEN
			fb_state_entry.i16_next_step := 50;
		END_IF

(*=======================================================*)
	50:	(* Änderungen im Camtable mit Eigenschaft: "mit sofortiger Wirkung" aktivieren *)
		IF fb_state_entry.E THEN
			mc_set_cam_online_change_mode.ActivationMode := MC_CAMACTIVATION_INSTANTANEOUS;
			mc_set_cam_online_change_mode.MasterScalingMode := MC_CAMSCALING_USERDEFINED;
			mc_set_cam_online_change_mode.SlaveScalingMode := MC_CAMSCALING_USERDEFINED;
			mc_set_cam_online_change_mode.CamTableID := 4;
			mc_set_cam_online_change_mode.Execute := TRUE;
		END_IF

		(*-----------------------Weiterschaltbedingungen----------------------------*)
		IF mc_set_cam_online_change_mode.Done THEN
			mc_set_cam_online_change_mode.Execute := FALSE;
			fb_state_entry.i16_next_step := 55;
		ELSIF mc_set_cam_online_change_mode.Error THEN
			err_id := mc_set_cam_online_change_mode.ErrorID;
			fb_state_entry.i16_next_step := FEHLER;
		END_IF

(*=======================================================*)
	55:	(* Überprüfe Nullpunktverschiebung des Absolutwertgebers auf Korrektheit *)
		IF fb_state_entry.E THEN
			fb_axis.i16_nc_parameter_nummer := AxisEncoderOffset;	(* vom Datentyp MC_AxisParameter *)
			st_drive_cmd.enu_cmd := READ_NC_PARAMETER;
		END_IF

		(*-----------------------Weiterschaltbedingungen----------------------------*)
		IF st_drive_cmd.enu_cmd = NO_COMMAND THEN
			IF fb_axis.r_wert_nc_read_parameter = gst_datensatz.st_md.st_md_b_achse.lr_nullpunktverschiebung THEN
				fb_state_entry.i16_next_step := 60;	(* Reglerfreigabe setzen *)
			ELSE
				fb_state_entry.i16_next_step := 56;	(* Nullpunktverschiebung schreiben *)
			END_IF
		END_IF

(*=======================================================*)
	56:	(* Nullpunktverschiebung hat sich geändert, deshalb erst Null reinschreiben, um keinen Additionsfehler zu machen, *)
		(* weil der Wert der Verschiebung beim Neustart komplett auf die Achse geschrieben wird *)
		IF fb_state_entry.E THEN
			fb_axis.i16_nc_parameter_nummer := AxisEncoderOffset;
			fb_axis.r_wert_nc_write_parameter := 0.0;
			st_drive_cmd.enu_cmd := WRITE_NC_PARAMETER;
		END_IF

		(*-----------------------Weiterschaltbedingungen----------------------------*)
		IF st_drive_cmd.enu_cmd = NO_COMMAND THEN
			fb_state_entry.i16_next_step := 57;
		END_IF

(*=======================================================*)
	57:	(* Aktuelle Nullpunktverschiebung des Absolutwertgebers an die Achse senden *)
		IF fb_state_entry.E THEN
			fb_axis.i16_nc_parameter_nummer := AxisEncoderOffset;
			fb_axis.r_wert_nc_write_parameter := gst_datensatz.st_md.st_md_b_achse.lr_nullpunktverschiebung;
			st_drive_cmd.enu_cmd := WRITE_NC_PARAMETER;
		END_IF

		(*-----------------------Weiterschaltbedingungen----------------------------*)
		IF st_drive_cmd.enu_cmd = NO_COMMAND THEN
			fb_state_entry.i16_next_step := 60;
		END_IF

(*=======================================================*)
	60:	(* Reglerfreigabe setzen , Reset wird bei Bedarf automatisch ausgeführt*)
		IF fb_state_entry.E THEN
			st_drive_cmd.enu_cmd := POWER_ENABLE;
		END_IF

		(*-----------------------Weiterschaltbedingungen----------------------------*)
		IF st_drive_cmd.enu_cmd = NO_COMMAND THEN
			fb_state_entry.i16_next_step := 70;
		END_IF

(*=======================================================*)
	70:	(* Nullpunktverschiebung ist geschrieben *)
		IF fb_state_entry.E THEN
			st_ctrl_out.b_prebereit := TRUE;
		END_IF

		(*-----------------------Weiterschaltbedingungen----------------------------*)
		IF st_ctrl_in.b_init THEN
			fb_state_entry.i16_next_step := BEREIT;
		END_IF

(*=======================================================*)
	BEREIT:
		IF fb_state_entry.E THEN
			b_referenzieren := FALSE;
			st_ctrl_out.b_bereit := TRUE;
		END_IF

		(*-----------------------Weiterschaltbedingungen----------------------------*)
		IF st_ctrl_in.b_bremse_auf THEN
			fb_state_entry.i16_next_step := 200;	(* Motorbremse lösen *)
		ELSIF st_ctrl_in.b_bremse_zu THEN
			fb_state_entry.i16_next_step := 300;	(* Motorbremse fest *)
		ELSIF st_ctrl_in.b_home THEN
			fb_state_entry.i16_next_step := 400;	(* HOME *)
			st_ctrl_out.b_fertig_2 := FALSE;
		ELSIF st_ctrl_in.b_start THEN
			st_ctrl_out.b_fertig := FALSE;
			st_ctrl_out.b_fertig_2 := FALSE;
			fb_state_entry.i16_next_step := 500;	(* Einfädelprozedur *)
		ELSIF st_ctrl_in.b_ausfaedeln_servo THEN
			fb_state_entry.i16_next_step := 700;	(* Band ausfädeln *)
		ELSIF st_ctrl_in.b_startpos THEN
			st_ctrl_out.b_servo_auf_einfaedelpos := FALSE;
			fb_state_entry.i16_next_step := 800; (*Igelrad auf Startposition fahren*)
		END_IF

(*=======================================================*)
	200:	(* Reglerfreigabe wegnehmen *)
		IF fb_state_entry.E THEN
			st_drive_cmd.enu_cmd := POWER_DISABLE;
		END_IF

		(*-----------------------Weiterschaltbedingungen----------------------------*)
		IF st_drive_cmd.enu_cmd = NO_COMMAND THEN
			fb_state_entry.i16_next_step := 210;
		END_IF

(*=======================================================*)
	210:	(* Motorbremse auf *)
		IF fb_state_entry.E THEN
			fb_axis.w_idn := P_0_IDN + 96;
			fb_axis.ui16_soeparam_write_value := 2;
			st_drive_cmd.enu_cmd := SOE_WRITE_PARAM;
		END_IF

		(*-----------------------Weiterschaltbedingungen----------------------------*)
		IF st_drive_cmd.enu_cmd = NO_COMMAND THEN
			fb_state_entry.i16_next_step := 220;
		END_IF

(*=======================================================*)
	220:	(* Fertig *)
		IF fb_state_entry.E THEN
			st_ctrl_out.b_bremse_geoeffnet := TRUE;
			fb_ton_wz.PT := t#50ms;
			fb_ton_wz.IN := TRUE;
		END_IF

		(*-----------------------Weiterschaltbedingungen----------------------------*)
		IF fb_ton_wz.Q THEN
			fb_ton_wz.IN := FALSE;
			st_ctrl_out.b_bremse_geoeffnet := FALSE;
			fb_state_entry.i16_next_step := BEREIT;
		END_IF

(*=======================================================*)
	300:	(* Reglerfreigabe setzen *)
		IF fb_state_entry.E THEN
			st_drive_cmd.enu_cmd := POWER_ENABLE;
		END_IF

		(*-----------------------Weiterschaltbedingungen----------------------------*)
		IF st_drive_cmd.enu_cmd = NO_COMMAND THEN
			st_ctrl_out.b_bremse_geschlossen := TRUE;
			(* Einzug wieder mit vollem Strom fahren *)
			i_Stromlimit := i16_max_torque;
			fb_state_entry.i16_next_step := 310;
		END_IF

(*=======================================================*)
	310:	(* Motorbremse zu *)
		IF fb_state_entry.E THEN
			fb_axis.w_idn := P_0_IDN + 96;
			fb_axis.ui16_soeparam_write_value := 0;
			st_drive_cmd.enu_cmd := SOE_WRITE_PARAM;
		END_IF

		(*-----------------------Weiterschaltbedingungen----------------------------*)
		IF st_drive_cmd.enu_cmd = NO_COMMAND THEN
			fb_state_entry.i16_next_step := 320;
		END_IF

(*=======================================================*)
	320:	(* Fertig *)
		IF fb_state_entry.E THEN
			st_ctrl_out.b_bremse_geschlossen := TRUE;
			fb_ton_wz.PT := t#50ms;
			fb_ton_wz.IN := TRUE;
		END_IF

		(*-----------------------Weiterschaltbedingungen----------------------------*)
		IF fb_ton_wz.Q THEN
			fb_ton_wz.IN := FALSE;
			st_ctrl_out.b_bremse_geschlossen := FALSE;
			fb_state_entry.i16_next_step := BEREIT;
		END_IF

(*=======================================================*)
	400:	(* HOME *)
		IF fb_state_entry.E THEN
			st_drive_cmd.enu_cmd := HOME;
		END_IF

		(*-----------------------Weiterschaltbedingungen----------------------------*)
		IF st_drive_cmd.enu_cmd = NO_COMMAND AND NOT fb_state_entry.E THEN
			st_ctrl_out.b_fertig_2 := TRUE;
			fb_state_entry.i16_next_step := 410;

			(* Torqueerst nach HOME wieder hoch nehmen *)
			lr_merker_pos_nach_lueften := b_achse.NcToPlc.ActPos;
			i_Stromlimit := i16_max_torque;
		
			lr_merker_pos_diff_lueften := lr_merker_pos_nach_lueften - lr_merker_pos_vor_lueften;
		END_IF

	410:
		IF NOT st_ctrl_in.b_home THEN
			st_ctrl_out.b_fertig_2 := FALSE;
			fb_state_entry.i16_next_step := BEREIT;
		END_IF

(*=======================================================*)
	500:(* Band von Bediener in das Igelrad einfädeln oder Vorschub ins Igelrad einfädeln *)
		IF fb_state_entry.E THEN
			fb_ton_wz.IN := FALSE;
		END_IF

		IF 	(zyl_bawe_querschub.fb.e_sensor1_eingefahren AND
			zyl_bawe_halter_li.st_ctrl.out.b_eingefahren AND
			zyl_bawe_faenger_li.st_ctrl.out.b_eingefahren AND
			(visu_hinten.out.ST_Servobandeinzug.b_taste_tippen OR
			st_ctrl_in.b_einfaedeln_servo)) OR
			(zyl_bawe_querschub.fb.e_sensor1_ausgefahren AND
			zyl_bawe_halter_re.st_ctrl.out.b_eingefahren AND
			zyl_bawe_faenger_re.st_ctrl.out.b_eingefahren AND
			(visu_hinten.out.ST_Servobandeinzug.b_taste_tippen OR
			st_ctrl_in.b_einfaedeln_servo))
			THEN
				fb_state_entry.i16_next_step := 531;
		END_IF

(*=======================================================*)
	531:(* Reglerfreigabe wegnehmen *)
		IF fb_state_entry.E THEN
			st_drive_cmd.enu_cmd := POWER_DISABLE;
		END_IF

		(*-----------------------Weiterschaltbedingungen----------------------------*)
		IF st_drive_cmd.enu_cmd = NO_COMMAND THEN
			fb_state_entry.i16_next_step :=533;
		END_IF

(*=======================================================*)
	533:	(* Reglerfreigabe setzen aktuelle Position wird Sollpositon*)
		IF fb_state_entry.E THEN
			st_drive_cmd.enu_cmd := POWER_ENABLE;
		END_IF

		(*-----------------------Weiterschaltbedingungen----------------------------*)
		IF st_drive_cmd.enu_cmd = NO_COMMAND THEN
			fb_state_entry.i16_next_step :=535;
		END_IF

(*=======================================================*)
	535:	(* Band fährt in GLS*)
		IF fb_state_entry.E THEN
			fb_axis.lr_soll_geschwindigkeit := st_geschwindigkeiten.lr_jog;
			(* Drehmoment hochsetzen *)
			i_Stromlimit := i16_man_einfaedel_torque;
			IF st_ctrl_in.b_einfaedeln_servo THEN
				fb_ton_uez.PT := t#10s;
				fb_ton_uez.IN := TRUE;
			END_IF
		END_IF

		st_drive_cmd.enu_cmd := JOG_VORWAERTS;

		(*-----------------------Weiterschaltbedingungen----------------------------*)
		IF e_gls_bandreferenzieren THEN
			fb_state_entry.i16_next_step := 540;
		END_IF

		IF fb_ton_uez.Q THEN
			sm_band_nicht_in_lichtschranke := TRUE;
			fb_state_entry.i16_next_step := FEHLER;
		END_IF

		IF fb_state_entry.X THEN
			fb_ton_uez.IN := FALSE;
		END_IF

(*=======================================================*)
	540:	(* Einzug Tippen Stop. *)
		IF fb_state_entry.E THEN
			st_drive_cmd.enu_cmd := JOG_STOP;
		END_IF

		(*-----------------------Weiterschaltbedingungen----------------------------*)
		IF st_drive_cmd.enu_cmd = NO_COMMAND THEN
			fb_state_entry.i16_next_step := 550;
		END_IF

(*=======================================================*)
	550:	(* Schleppabstandsüberwachung einschalten. *)
		IF fb_state_entry.E THEN
			i_Stromlimit := i16_auto_einfaedel_torque;
			fb_axis.i16_nc_parameter_nummer := EnablePosLagMonitoring;
			fb_axis.r_wert_nc_write_parameter := 1;
			st_drive_cmd.enu_cmd := WRITE_NC_PARAMETER;
		END_IF

		(*-----------------------Weiterschaltbedingungen----------------------------*)
		IF st_drive_cmd.enu_cmd = NO_COMMAND THEN
			fb_state_entry.i16_next_step := 560;
		END_IF

(*=======================================================*)
	560:	(* Band zurück bis GLS sicher aus (Sicherstellen das das Band an der Richtigen Position startet) *)
		IF fb_state_entry.E THEN
			st_drive_cmd.enu_cmd := MOVE_RELATIVE;
			fb_axis.lr_soll_geschwindigkeit := st_geschwindigkeiten.lr_jog;
			fb_axis.st_position.r_soll := F_Servobandeinzug_Strecke_zu_Grad( strecke := - lr_max_strecke_gls_wkz);
		END_IF

		(*-----------------------Weiterschaltbedingungen----------------------------*)
		IF st_drive_cmd.enu_cmd = NO_COMMAND THEN
			(* Zielposition wurde erreicht -> kein korrekter Abschluss *)
			fb_state_entry.i16_next_step := FEHLER;
			sm_bandrueckzug := TRUE;
		ELSIF NOT fb_tof_gls_ref.Q THEN
			fb_state_entry.i16_next_step := 570;
		END_IF

(*=======================================================*)
	570:
		IF fb_state_entry.E THEN
			st_drive_cmd.enu_cmd := STOP_AXIS;
		END_IF

		(*-----------------------Weiterschaltbedingungen----------------------------*)
		IF st_drive_cmd.enu_cmd = NO_COMMAND THEN
			fb_state_entry.i16_next_step := 580;
		END_IF

(*=======================================================*)
	580: (* Fahre Band langsam bis zur GLS *)
		IF fb_state_entry.E THEN
			st_drive_cmd.enu_cmd := MOVE_RELATIVE;
			fb_axis.lr_soll_geschwindigkeit := 0.2 * st_geschwindigkeiten.lr_jog;
			fb_axis.st_position.r_soll :=  F_Servobandeinzug_Strecke_zu_Grad( strecke := lr_max_strecke_gls_wkz );
		END_IF

		(*-----------------------Weiterschaltbedingungen----------------------------*)
		IF st_drive_cmd.enu_cmd = NO_COMMAND THEN
			(* Zielposition wurde erreicht -> kein korrekter Abschluss *)
			fb_state_entry.i16_next_step := FEHLER;
			sm_fahren_auf_gls := TRUE;
		ELSIF e_gls_bandreferenzieren THEN
			fb_state_entry.i16_next_step := 590;
		END_IF

(*=======================================================*)
	590:
		IF fb_state_entry.E THEN
			st_drive_cmd.enu_cmd := STOP_AXIS;
		END_IF

		(*-----------------------Weiterschaltbedingungen----------------------------*)
		IF st_drive_cmd.enu_cmd = NO_COMMAND THEN
			fb_state_entry.i16_next_step := 600;
		END_IF

(*=======================================================*)
	600:	(* Band bis zum ersten Fänger im WKZ  fahren - Unterteilung in 2 Wegstrecken mit 2 Geschwindigkeiten. *)
		IF fb_state_entry.E THEN
			fb_axis.lr_soll_geschwindigkeit := st_geschwindigkeiten.lr_jog;
			fb_axis.st_position.r_soll := F_Servobandeinzug_Strecke_zu_Grad( strecke := lr_konst_strecke_ls_bandeinzug );
			st_drive_cmd.enu_cmd := MOVE_RELATIVE;
		END_IF

		(*-----------------------Weiterschaltbedingungen----------------------------*)
		IF st_drive_cmd.enu_cmd = NO_COMMAND THEN
			fb_state_entry.i16_next_step := 605;
		END_IF

(*=======================================================*)
	605:	(* Schleppabstandsüberwachung ausschalten *)
		IF fb_state_entry.E THEN
			fb_axis.i16_nc_parameter_nummer := EnablePosLagMonitoring;
			fb_axis.r_wert_nc_write_parameter := 0;
			st_drive_cmd.enu_cmd := WRITE_NC_PARAMETER;
		END_IF

		(*-----------------------Weiterschaltbedingungen----------------------------*)
		IF st_drive_cmd.enu_cmd = NO_COMMAND THEN
			fb_state_entry.i16_next_step := 610;
		END_IF

(*=======================================================*)
	610:	(* Band bis zum ersten Fänger im WKZ  fahren *)
		IF fb_state_entry.E THEN
			fb_axis.lr_soll_geschwindigkeit := 0.2 * st_geschwindigkeiten.lr_jog;
			fb_axis.st_position.r_soll :=  F_Servobandeinzug_Strecke_zu_Grad( strecke := lr_max_strecke_gls_wkz - lr_konst_strecke_ls_bandeinzug );
			st_drive_cmd.enu_cmd := MOVE_RELATIVE;
		END_IF

		(*-----------------------Weiterschaltbedingungen----------------------------*)
		IF st_drive_cmd.enu_cmd = NO_COMMAND THEN
			(* Zielposition wurde erreicht -> kein korrekter Abschluss *)
			sm_fehler_bandeinfaedeln := TRUE;
			st_drive_cmd.enu_cmd := STOP_AXIS;
			fb_state_entry.i16_next_step := FEHLER;
		ELSIF ABS(i16_torque) > i16_block_torque THEN
			(* Wenn Strom steigt, dann steht Band an Fänger im WKZ an. *)
			fb_state_entry.i16_next_step := 620;
		END_IF

(*=======================================================*)
	620:	(* Einzug STOP - Einfädelprozedur beendet. *)
		IF fb_state_entry.E THEN
			st_drive_cmd.enu_cmd := STOP_AXIS;
		END_IF

		(*-----------------------Weiterschaltbedingungen----------------------------*)
		IF st_drive_cmd.enu_cmd = NO_COMMAND THEN
			fb_state_entry.i16_next_step := 630;
		END_IF

(*=======================================================*)
	630:	(* Antrieb kurzfristig kraftlos schalten zum Bandlüften. *)
		IF fb_state_entry.E THEN
			fb_ton_wz.PT := t#1000ms;
			fb_ton_wz.IN := TRUE;
			i_Stromlimit := i16_einfaedel_torque;
		END_IF

		(*-----------------------Weiterschaltbedingungen----------------------------*)
		IF fb_ton_wz.Q THEN
			fb_ton_wz.IN := FALSE;
			fb_state_entry.i16_next_step := 640;
		END_IF

(*=======================================================*)
	640: (* Warte kurz *)
		IF fb_state_entry.E THEN
			fb_ton_wz.PT := t#1000ms;
			fb_ton_wz.IN := TRUE;
		END_IF

		(*-----------------------Weiterschaltbedingungen----------------------------*)
		IF fb_ton_wz.Q THEN
			fb_ton_wz.IN := FALSE;
			fb_state_entry.i16_next_step := 650;
		END_IF

(*=======================================================*)
	650:	(* Position nullen *)
		IF fb_state_entry.E THEN
			st_drive_cmd.enu_cmd := HOME;
		END_IF

		(*-----------------------Weiterschaltbedingungen----------------------------*)
		IF st_drive_cmd.enu_cmd = NO_COMMAND THEN
			(* Volles Drehmoment *)
			i_Stromlimit := i16_max_torque;
			fb_state_entry.i16_next_step := 660;
		END_IF

(*=======================================================*)
	660:	(* Schleppabstandsüberwachung wieder einschalten *)
		IF fb_state_entry.E THEN
			fb_axis.i16_nc_parameter_nummer := EnablePosLagMonitoring;
			fb_axis.r_wert_nc_write_parameter := 1;
			st_drive_cmd.enu_cmd := WRITE_NC_PARAMETER;
		END_IF

		(*-----------------------Weiterschaltbedingungen----------------------------*)
		IF st_drive_cmd.enu_cmd = NO_COMMAND THEN
			st_ctrl_out.b_fertig := TRUE;
			fb_state_entry.i16_next_step := BEREIT;
		END_IF

(*=======================================================*)
	700:	(* Band ausfädeln, damit der Ausschiebezylinder sicher trifft. *)
		IF fb_state_entry.E THEN
			i_Stromlimit := i16_auto_einfaedel_torque;(*i16_max_torque*)
			fb_axis.lr_soll_geschwindigkeit := 0.2 * st_geschwindigkeiten.lr_jog;
			fb_axis.st_position.r_soll :=  F_Servobandeinzug_Strecke_zu_Grad( strecke := - gst_datensatz.st_band.r_raster * 93);
			st_drive_cmd.enu_cmd := MOVE_RELATIVE;
		END_IF

		(*-----------------------Weiterschaltbedingungen----------------------------*)
		IF st_drive_cmd.enu_cmd = NO_COMMAND THEN
			fb_state_entry.i16_next_step := 705;
		END_IF

(*=======================================================*)
	705:	(* Schleppabstandsüberwachung ausschalten *)
		IF fb_state_entry.E THEN
			fb_axis.i16_nc_parameter_nummer := EnablePosLagMonitoring;
			fb_axis.r_wert_nc_write_parameter := 0;
			st_drive_cmd.enu_cmd := WRITE_NC_PARAMETER;
		END_IF

		(*-----------------------Weiterschaltbedingungen----------------------------*)
		IF st_drive_cmd.enu_cmd = NO_COMMAND THEN
			fb_state_entry.i16_next_step := 710;
		END_IF

(*=======================================================*)
	710:	(* Fertig *)
		IF fb_state_entry.E THEN
(*			i_Stromlimit := 25;(*Neu*)*)
			st_ctrl_out.b_ausgefaedelt_servo := TRUE;
			fb_ton_wz.PT := t#50ms;
			fb_ton_wz.IN := TRUE;
		END_IF

		(*-----------------------Weiterschaltbedingungen----------------------------*)
		IF fb_ton_wz.Q THEN
			fb_ton_wz.IN := FALSE;
			st_ctrl_out.b_ausgefaedelt_servo := FALSE;
			fb_state_entry.i16_next_step := BEREIT;
		END_IF

(*=======================================================*)
	800:	(* Reglerfreigabe setzen *)
		IF fb_state_entry.E THEN
			st_drive_cmd.enu_cmd := POWER_ENABLE;
		END_IF

		(*-----------------------Weiterschaltbedingungen----------------------------*)
		IF st_drive_cmd.enu_cmd = NO_COMMAND THEN
			fb_state_entry.i16_next_step :=810;
		END_IF

(*=======================================================*)
	810:	(* Bremse automatisch *)
		IF fb_state_entry.E THEN
			fb_axis.w_idn := P_0_IDN + 96;
			fb_axis.ui16_soeparam_write_value := 0;
			st_drive_cmd.enu_cmd := SOE_WRITE_PARAM;
		END_IF

		(*-----------------------Weiterschaltbedingungen----------------------------*)
		IF st_drive_cmd.enu_cmd = NO_COMMAND THEN
			fb_state_entry.i16_next_step := 820;
		END_IF

(*=======================================================*)
	820:	(* Startposition Igelrad berechnen *)
		IF fb_state_entry.E THEN
			lr_startpos :=  F_Startpos_Servobandeinzug( r_actual_pos := b_achse.NcToPlc.ModuloActPos);
			IF lr_startpos < b_achse.NcToPlc.ModuloActPos THEN
				fb_axis.st_position.r_soll :=  lr_startpos - b_achse.NcToPlc.ModuloActPos;
			ELSE
				fb_axis.st_position.r_soll := b_achse.NcToPlc.ModuloActPos - lr_startpos ;
			END_IF
		END_IF

		(*-----------------------Weiterschaltbedingungen----------------------------*)
		fb_state_entry.i16_next_step := 830;

(*=======================================================*)
	830: (* Positioniere Achse auf Einfädelposition *)
		IF fb_state_entry.E THEN
			i_Stromlimit := i16_max_torque;
			fb_axis.lr_soll_geschwindigkeit := st_geschwindigkeiten.lr_jog;
			st_drive_cmd.enu_cmd := MOVE_RELATIVE;
		END_IF

		(*-----------------------Weiterschaltbedingungen----------------------------*)
		IF st_drive_cmd.enu_cmd = NO_COMMAND THEN
			fb_state_entry.i16_next_step := 840;
		END_IF

(*=======================================================*)
	840:	(* Schleppabstandsüberwachung ausschalten *)
		IF fb_state_entry.E THEN
			fb_axis.i16_nc_parameter_nummer := EnablePosLagMonitoring;
			fb_axis.r_wert_nc_write_parameter := 0;
			st_drive_cmd.enu_cmd := WRITE_NC_PARAMETER;
		END_IF

		(*-----------------------Weiterschaltbedingungen----------------------------*)
		IF st_drive_cmd.enu_cmd = NO_COMMAND THEN
			fb_state_entry.i16_next_step := 850;
		END_IF

(*=======================================================*)
	850:	(* Drehmoment auf ein Minimum begrenzen zum Einfädeln *)
		IF fb_state_entry.E THEN
			(* Drehmoment auf Minimum reduzieren *)
			i_Stromlimit := i16_lueft_torque;
		END_IF

		(*-----------------------Weiterschaltbedingungen----------------------------*)
		fb_state_entry.i16_next_step := BEREIT;
		st_ctrl_out.b_servo_auf_einfaedelpos := TRUE;

(*=======================================================*)
	FEHLER:
		IF fb_state_entry.E THEN
			st_ctrl_out.b_fehler := TRUE;
			fb_ton_quitt.IN := FALSE;
		END_IF

		(* =====Achse wird gestoppt===== *)
		IF st_ctrl_in.b_stop AND NOT b_achse.Status.HasBeenStopped THEN
			st_drive_cmd.enu_cmd := STOP_AXIS;

		(* =====Achse wird angehalten===== *)
		ELSIF st_ctrl_in.b_halt AND NOT b_achse.Status.NotMoving THEN
			st_drive_cmd.enu_cmd := HALT_AXIS;
		END_IF

		(*-----------------------Weiterschaltbedingungen----------------------------*)
		IF st_ctrl_in.b_quitt AND NOT fb_state_entry.E THEN
			st_ctrl_out.b_fehler := FALSE;
			st_drive_cmd.enu_cmd := RESET;
			fb_ton_quitt.IN := TRUE;
		END_IF

		IF fb_ton_quitt.Q THEN
			fb_ton_quitt.IN := FALSE;
			fb_state_entry.i16_next_step := INIT;
		END_IF

(*=======================================================*)
	STOP:
		IF fb_state_entry.E THEN
			IF b_achse.NcToPlc.CoupleState = 0 THEN
				st_drive_cmd.enu_cmd := STOP_AXIS;
			END_IF
			fb_ton_quitt.IN := FALSE;
		END_IF

		(*-----------------------Weiterschaltbedingungen----------------------------*)
		IF st_drive_cmd.enu_cmd = NO_COMMAND AND b_achse.Status.NotMoving THEN
			fb_state_entry.i16_next_step := STILLSTAND;
		END_IF

(*=======================================================*)
	STILLSTAND:
		IF fb_state_entry.E THEN
			st_drive_cmd.enu_cmd := POWER_DISABLE;
			fb_ton_quitt.IN := FALSE;
		END_IF

		(*-----------------------Weiterschaltbedingungen----------------------------*)
		IF st_ctrl_in.b_quitt AND NOT fb_state_entry.E THEN
			fb_ton_quitt.IN := TRUE;
		END_IF

		IF fb_ton_quitt.Q THEN
			fb_ton_quitt.IN := FALSE;
			fb_state_entry.i16_next_step := INIT;
		END_IF

(*=======================================================*)
	HALT:
		IF fb_state_entry.E THEN
			IF b_achse.NcToPlc.CoupleState = 0 THEN
				st_drive_cmd.enu_cmd := HALT_AXIS;
			END_IF
			fb_ton_quitt.IN := FALSE;
		END_IF

		(*-----------------------Weiterschaltbedingungen----------------------------*)
		IF st_ctrl_in.b_quitt AND NOT fb_state_entry.E THEN
			fb_ton_quitt.IN := TRUE;
		END_IF

		IF fb_ton_quitt.Q THEN
			fb_ton_quitt.IN := FALSE;
			fb_state_entry.i16_next_step := INIT;
		END_IF

(*=======================================================*)
	HANDRAD:
		IF fb_state_entry.E THEN
			st_ctrl_out.b_fehler := TRUE;
			fb_axis.lr_soll_geschwindigkeit := st_geschwindigkeiten.lr_jog;
			i_Stromlimit := i16_max_torque / 2;
		END_IF


		IF 	zyl_bawe_querschub.fb.e_sensor1_eingefahren AND
			zyl_bawe_halter_li.st_ctrl.out.b_eingefahren AND
			zyl_bawe_faenger_li.st_ctrl.out.b_eingefahren
			THEN
				IF ST_Euchner_Handbedienpult.i16_Handrad_delta > 0 THEN
					st_drive_cmd.enu_cmd := JOG_VORWAERTS;
				END_IF
				IF ST_Euchner_Handbedienpult.i16_Handrad_delta < 0 THEN
						st_drive_cmd.enu_cmd := JOG_RUECKWAERTS;
				END_IF
		ELSIF 	zyl_bawe_querschub.fb.e_sensor1_ausgefahren AND
				zyl_bawe_halter_re.st_ctrl.out.b_eingefahren AND
				zyl_bawe_faenger_re.st_ctrl.out.b_eingefahren
				THEN
					IF ST_Euchner_Handbedienpult.i16_Handrad_delta > 0 THEN
						st_drive_cmd.enu_cmd := JOG_VORWAERTS;
					END_IF
					IF ST_Euchner_Handbedienpult.i16_Handrad_delta < 0 THEN
							st_drive_cmd.enu_cmd := JOG_RUECKWAERTS;
					END_IF
		ELSE
			IF b_achse.Status.Moving THEN
				st_drive_cmd.enu_cmd := JOG_STOP;
			END_IF
		END_IF

		IF fb_r_trig_taste_plus.Q THEN
			fb_state_entry.i16_next_step := MOTORBREMSE_AUF;
		END_IF
		IF fb_r_trig_taste_minus.Q THEN
			fb_state_entry.i16_next_step := MOTORBREMSE_ZU;
		END_IF

		(*-----------------------Weiterschaltbedingungen----------------------------*)
		IF gi16_betriebsart <> HAND OR NOT b_hand_dialog_aktiv THEN
			fb_state_entry.i16_next_step := 2010;
		END_IF

(*=======================================================*)
	2010:
		IF fb_state_entry.E THEN
			st_drive_cmd.enu_cmd := ABORT;
		END_IF

		(*-----------------------Weiterschaltbedingungen----------------------------*)
		IF st_drive_cmd.enu_cmd = NO_COMMAND THEN
			fb_state_entry.i16_next_step := 2020;
		END_IF

(*=======================================================*)
	2020:
		IF fb_state_entry.E THEN
			fb_axis.w_idn := P_0_IDN + 96;
			fb_axis.ui16_soeparam_write_value := 0;
			st_drive_cmd.enu_cmd := SOE_WRITE_PARAM;
		END_IF

		(*-----------------------Weiterschaltbedingungen----------------------------*)
		IF st_drive_cmd.enu_cmd = NO_COMMAND THEN
			fb_state_entry.i16_next_step := 2030;
		END_IF

(*=======================================================*)
	2030:	(* Reglerfreigabe wegnehmen *)
		IF fb_state_entry.E THEN
			st_drive_cmd.enu_cmd := POWER_DISABLE;
		END_IF

		(*-----------------------Weiterschaltbedingungen----------------------------*)
		IF st_drive_cmd.enu_cmd = NO_COMMAND THEN
			st_ctrl_out.b_fehler := FALSE;
			fb_state_entry.i16_next_step := INIT;
		END_IF

(*=======================================================*)
	MOTORBREMSE_AUF:
		IF fb_state_entry.E THEN
			st_drive_cmd.enu_cmd := ABORT;
		END_IF

		(*-----------------------Weiterschaltbedingungen----------------------------*)
		IF st_drive_cmd.enu_cmd = NO_COMMAND THEN
			fb_state_entry.i16_next_step := 2110;
		END_IF

(*=======================================================*)
	2110:	(* Reglerfreigabe wegnehmen *)
		IF fb_state_entry.E THEN
			st_drive_cmd.enu_cmd := POWER_DISABLE;
		END_IF

		(*-----------------------Weiterschaltbedingungen----------------------------*)
		IF st_drive_cmd.enu_cmd = NO_COMMAND THEN
			fb_state_entry.i16_next_step := 2120;
		END_IF

(*=======================================================*)
	2120:	(* Bremse auf machen *)
		IF fb_state_entry.E THEN
			fb_axis.w_idn := P_0_IDN + 96;
			fb_axis.ui16_soeparam_write_value := 2;
			st_drive_cmd.enu_cmd := SOE_WRITE_PARAM;
		END_IF

		(*-----------------------Weiterschaltbedingungen----------------------------*)
		IF 	st_drive_cmd.enu_cmd = NO_COMMAND AND
			(gi16_betriebsart <> HAND OR
			NOT b_hand_dialog_aktiv OR
			ST_Euchner_Handbedienpult.i16_Handrad_delta > 0)
			THEN
				fb_state_entry.i16_next_step := HANDRAD;
		ELSIF fb_r_trig_taste_minus.Q THEN
			fb_state_entry.i16_next_step := MOTORBREMSE_ZU;
		END_IF

(*=======================================================*)
	MOTORBREMSE_ZU:
		IF fb_state_entry.E THEN
			st_drive_cmd.enu_cmd := ABORT;
		END_IF

		(*-----------------------Weiterschaltbedingungen----------------------------*)
		IF st_drive_cmd.enu_cmd = NO_COMMAND THEN
			fb_state_entry.i16_next_step := 2210;
		END_IF

(*=======================================================*)
	2210:	(* Reglerfreigabe setzen *)
		IF fb_state_entry.E THEN
			st_drive_cmd.enu_cmd := POWER_ENABLE;
		END_IF

		(*-----------------------Weiterschaltbedingungen----------------------------*)
		IF st_drive_cmd.enu_cmd = NO_COMMAND THEN
			fb_state_entry.i16_next_step := 2220;
		END_IF

(*=======================================================*)
	2220:	(* Bremse zu machen *)
		IF fb_state_entry.E THEN
			fb_axis.w_idn := P_0_IDN + 96;
			fb_axis.ui16_soeparam_write_value := 0;
			st_drive_cmd.enu_cmd := SOE_WRITE_PARAM;
		END_IF

		(*-----------------------Weiterschaltbedingungen----------------------------*)
		IF 	st_drive_cmd.enu_cmd = NO_COMMAND AND
			(gi16_betriebsart <> HAND OR
			NOT b_hand_dialog_aktiv OR
			ST_Euchner_Handbedienpult.i16_Handrad_delta > 0)
			THEN
				fb_state_entry.i16_next_step := HANDRAD;
		ELSIF fb_r_trig_taste_plus.Q THEN
			fb_state_entry.i16_next_step := MOTORBREMSE_AUF;
		END_IF

(*=======================================================*)
	LUEFTEN:
		IF fb_state_entry.E THEN
			st_drive_cmd.enu_cmd := POWER_DISABLE;
			fb_ton_wz_disable.IN := TRUE;
			fb_ton_quitt.IN := FALSE;
		END_IF

		IF fb_ton_wz_disable.Q AND st_drive_cmd.enu_cmd = NO_COMMAND THEN
			fb_axis.w_idn := P_0_IDN + 96;
			fb_axis.ui16_soeparam_write_value := 2;
			st_drive_cmd.enu_cmd := SOE_WRITE_PARAM;
			fb_ton_wz_disable.IN := FALSE;
		END_IF

		(*-----------------------Weiterschaltbedingungen----------------------------*)
		IF st_ctrl_in.b_quitt AND NOT fb_state_entry.E THEN
			fb_ton_wz_disable.IN := FALSE;
			fb_ton_quitt.IN := TRUE;
		END_IF

		IF fb_ton_quitt.Q THEN
			fb_ton_quitt.IN := FALSE;
			fb_state_entry.i16_next_step := INIT;
		END_IF

(*=======================================================*)
	REGELN:
		IF fb_state_entry.E THEN
			fb_ton_quitt.IN := FALSE;
			fb_axis.w_idn := P_0_IDN + 96;
			fb_axis.ui16_soeparam_write_value := 0;
			st_drive_cmd.enu_cmd := SOE_WRITE_PARAM;
		END_IF

		(*-----------------------Weiterschaltbedingungen----------------------------*)
		IF st_ctrl_in.b_quitt AND NOT fb_state_entry.E THEN
			fb_ton_wz_disable.IN := FALSE;
			fb_ton_quitt.IN := TRUE;
		END_IF

		IF fb_ton_quitt.Q THEN
			fb_ton_quitt.IN := FALSE;
			fb_state_entry.i16_next_step := INIT;
		END_IF

(*=======================================================*)
	INBETRIEBNAHME:	(* Überprüfe Nullpunktverschiebung des Absolutwertgebers auf Korrektheit *)
		IF fb_state_entry.E THEN
			fb_axis.i16_nc_parameter_nummer := AxisEncoderOffset;
			st_drive_cmd.enu_cmd := READ_NC_PARAMETER;
		END_IF

		(*-----------------------Weiterschaltbedingungen----------------------------*)
		IF st_drive_cmd.enu_cmd = NO_COMMAND THEN
			IF fb_axis.r_wert_nc_read_parameter = gst_datensatz.st_md.st_md_b_achse.lr_nullpunktverschiebung THEN
				fb_state_entry.i16_next_step := 5100;	(* Reversiersequenz*)
			ELSE
				fb_state_entry.i16_next_step := 5010;	(* Reglerfreigabe nehmen und Nullpunktverschiebung schreiben *)
			END_IF
		END_IF

(*=======================================================*)
	5010:	(* Reglerfreigabe wegnehmen, damit Nullpunktverschiebung geschrieben werden kannt*)
		IF fb_state_entry.E THEN
			st_drive_cmd.enu_cmd := POWER_DISABLE;
		END_IF

		(*-----------------------Weiterschaltbedingungen----------------------------*)
		IF st_drive_cmd.enu_cmd = NO_COMMAND THEN
			fb_state_entry.i16_next_step := 5020;
		END_IF

(*=======================================================*)
	5020:	(* Nullpunktverschiebung hat sich geändert, deshalb erst Null reinschreiben, um keinen Additionsfehler zu machen, *)
			(* weil der Wert der Verschiebung beim Neustart komplett auf die Achse geschrieben wird *)
		IF fb_state_entry.E THEN
			fb_axis.i16_nc_parameter_nummer := AxisEncoderOffset;
			fb_axis.r_wert_nc_write_parameter := 0.0;
			st_drive_cmd.enu_cmd := WRITE_NC_PARAMETER;
		END_IF

		(*-----------------------Weiterschaltbedingungen----------------------------*)
		IF st_drive_cmd.enu_cmd = NO_COMMAND THEN
			fb_state_entry.i16_next_step := 5030;
		END_IF

(*=======================================================*)
	5030:	(* Aktuelle Nullpunktverschiebung des Absolutwertgebers an die Achse senden *)
		IF fb_state_entry.E THEN
			fb_axis.i16_nc_parameter_nummer := AxisEncoderOffset;
			fb_axis.r_wert_nc_write_parameter := gst_datensatz.st_md.st_md_b_achse.lr_nullpunktverschiebung;
			st_drive_cmd.enu_cmd := WRITE_NC_PARAMETER;
		END_IF

		(*-----------------------Weiterschaltbedingungen----------------------------*)
		IF st_drive_cmd.enu_cmd = NO_COMMAND THEN
			fb_state_entry.i16_next_step := 5100;
		END_IF

(*=======================================================*)
	5100:	(* Verfahren der Achse zwischen zwei Punkten zum Testen verschiedener Achsparameter *)		(* Achse wird genullt *)
		IF fb_state_entry.E THEN
			st_drive_cmd.enu_cmd := HOME;
		END_IF

		(*-----------------------Weiterschaltbedingungen----------------------------*)
		IF st_drive_cmd.enu_cmd = NO_COMMAND THEN
			fb_state_entry.i16_next_step := 5110;
		END_IF

(*=======================================================*)
	5110:	(* Warte Start *)
		IF fb_state_entry.E THEN
			fb_axis.lr_soll_geschwindigkeit := st_geschwindigkeiten.lr_jog;
			fb_axis.st_position.lr_ibn_pos_ziel := 10.0;
		END_IF

		(*-----------------------Weiterschaltbedingungen----------------------------*)
		IF st_ctrl_in.b_ibn_start THEN
			fb_state_entry.i16_next_step := 5120;
		END_IF

(*=======================================================*)
	5120: (* Fahre Z-Achse auf Zielposition *)
		IF fb_state_entry.E THEN
			st_drive_cmd.enu_cmd := POWER_ENABLE;
		END_IF

		(*-----------------------Weiterschaltbedingungen----------------------------*)
		IF st_drive_cmd.enu_cmd = NO_COMMAND THEN
			;
		END_IF

(*=======================================================*)
	5130: (* Pause *)
		IF fb_state_entry.E THEN
			fb_ton_wz.PT := t#500ms;
			fb_ton_wz.IN := TRUE;
		END_IF

		(*-----------------------Weiterschaltbedingungen----------------------------*)
		IF fb_ton_wz.Q THEN
			fb_ton_wz.IN := FALSE;
			fb_state_entry.i16_next_step := 5110;
		END_IF
END_CASE

fb_state_entry(
	i16_next_step:= ,
	i16_pos:= 2,
	s_debugtext:= ,
	E=> ,
	X=> ,
	i16_step=> ,
	i16_last_step=> );

mc_set_cam_online_change_mode(
	Execute:= , 
	ActivationMode:= , 
	ActivationPosition:= , 
	MasterScalingMode:= , 
	SlaveScalingMode:= ,
	CamTableID:= ,
	Done=> , 
	Busy=> , 
	Error=> , 
	ErrorID=> );

IF st_config_achse.b_config_fertig THEN
	(* Fehlermeldungen und Betriebsmeldungen ab dem Startindex in die globalen Meldungsarrays schreiben *)
	garr_stoermeldungen[st_config_achse.i16_meld_startindex + 0] := st_sm.b_achse_nicht_bb;
	garr_stoermeldungen[st_config_achse.i16_meld_startindex + 1] := st_sm.b_achse_nicht_referenziert;
	garr_stoermeldungen[st_config_achse.i16_meld_startindex + 2] := st_sm.b_keine_verfahrfreigabe;
	garr_stoermeldungen[st_config_achse.i16_meld_startindex + 3] := st_sm.b_achse_nicht_auf_startpos;
	garr_stoermeldungen[st_config_achse.i16_meld_startindex + 4] := st_sm.b_ende_skalierungs_nocke;
	garr_stoermeldungen[st_config_achse.i16_meld_startindex + 5] := st_sm.b_ende_camming_nocke;
	garr_stoermeldungen[st_config_achse.i16_meld_startindex + 6] := st_sm.b_skalierung_noch_aktiv;
	garr_stoermeldungen[st_config_achse.i16_meld_startindex + 7] := FALSE;
	garr_stoermeldungen[st_config_achse.i16_meld_startindex + 8] := sm_bandrueckzug;
	garr_stoermeldungen[st_config_achse.i16_meld_startindex + 9] := sm_bandreferenzieren;
	garr_stoermeldungen[st_config_achse.i16_meld_startindex + 10] := sm_fehler_bandvorschub;
	garr_stoermeldungen[st_config_achse.i16_meld_startindex + 11] := sm_fehler_raster;
	garr_stoermeldungen[st_config_achse.i16_meld_startindex + 12] := sm_fehler_bandeinfaedeln;
	garr_stoermeldungen[st_config_achse.i16_meld_startindex + 13] := sm_fahren_auf_gls;
	garr_stoermeldungen[st_config_achse.i16_meld_startindex + 14] := sm_band_rausgezogen;
	garr_stoermeldungen[st_config_achse.i16_meld_startindex + 15] := sm_band_nicht_in_lichtschranke;
	garr_stoermeldungen[st_config_achse.i16_meld_startindex + 16] := st_drive_cmd.meldungen.sm_write_soe_parameter;
	garr_stoermeldungen[st_config_achse.i16_meld_startindex + 17] := st_drive_cmd.meldungen.sm_read_soe_parameter;
	garr_stoermeldungen[st_config_achse.i16_meld_startindex + 18] := st_drive_cmd.meldungen.sm_write_nc_parameter;
	garr_stoermeldungen[st_config_achse.i16_meld_startindex + 19] := st_drive_cmd.meldungen.sm_read_nc_parameter;
	garr_stoermeldungen[st_config_achse.i16_meld_startindex + 20] := st_drive_cmd.meldungen.sm_power_enable;
	garr_stoermeldungen[st_config_achse.i16_meld_startindex + 21] := st_drive_cmd.meldungen.sm_power_disable;
	garr_stoermeldungen[st_config_achse.i16_meld_startindex + 22] := st_drive_cmd.meldungen.sm_reset;
	garr_stoermeldungen[st_config_achse.i16_meld_startindex + 23] := st_drive_cmd.meldungen.sm_home;
	garr_stoermeldungen[st_config_achse.i16_meld_startindex + 24] := st_drive_cmd.meldungen.sm_setposition;
	garr_stoermeldungen[st_config_achse.i16_meld_startindex + 25] := st_drive_cmd.meldungen.sm_jog_vorwaerts;
	garr_stoermeldungen[st_config_achse.i16_meld_startindex + 26] := st_drive_cmd.meldungen.sm_jog_rueckwaerts;
	garr_stoermeldungen[st_config_achse.i16_meld_startindex + 27] := st_drive_cmd.meldungen.sm_move_absolute;
	garr_stoermeldungen[st_config_achse.i16_meld_startindex + 28] := st_drive_cmd.meldungen.sm_move_relative;
	garr_stoermeldungen[st_config_achse.i16_meld_startindex + 29] := st_drive_cmd.meldungen.sm_move_velocity;
	garr_stoermeldungen[st_config_achse.i16_meld_startindex + 30] := st_drive_cmd.meldungen.sm_move_modulo;
	garr_stoermeldungen[st_config_achse.i16_meld_startindex + 31] := st_drive_cmd.meldungen.sm_stop_axis;
	garr_stoermeldungen[st_config_achse.i16_meld_startindex + 32] := st_drive_cmd.meldungen.sm_halt_axis;
	garr_stoermeldungen[st_config_achse.i16_meld_startindex + 33] := st_drive_cmd.meldungen.sm_motion_command_timeout;
	garr_stoermeldungen[st_config_achse.i16_meld_startindex + 34] := st_sm.b_achsfehler;
	garr_stoermeldungen[st_config_achse.i16_meld_startindex + 35] := st_sm.b_devicefehler;
	garr_stoermeldungen[st_config_achse.i16_meld_startindex + 36] := st_drive_cmd.meldungen.sm_limit_positiv_erreicht;
	garr_stoermeldungen[st_config_achse.i16_meld_startindex + 37] := st_drive_cmd.meldungen.sm_limit_negativ_erreicht;
	garr_stoermeldungen[st_config_achse.i16_meld_startindex + 38] := st_drive_cmd.meldungen.sm_ec_coe_sdo_write_ex;
	garr_stoermeldungen[st_config_achse.i16_meld_startindex + 39] := st_drive_cmd.meldungen.sm_ec_coe_sdo_read_ex;
	garr_stoermeldungen[st_config_achse.i16_meld_startindex + 40] := FALSE;
	garr_stoermeldungen[st_config_achse.i16_meld_startindex + 41] := FALSE;
	garr_stoermeldungen[st_config_achse.i16_meld_startindex + 42] := FALSE;
	garr_stoermeldungen[st_config_achse.i16_meld_startindex + 43] := FALSE;
	garr_stoermeldungen[st_config_achse.i16_meld_startindex + 44] := FALSE;
	garr_stoermeldungen[st_config_achse.i16_meld_startindex + 45] := FALSE;
	garr_stoermeldungen[st_config_achse.i16_meld_startindex + 46] := FALSE;
	garr_stoermeldungen[st_config_achse.i16_meld_startindex + 47] := FALSE;
	garr_stoermeldungen[st_config_achse.i16_meld_startindex + 49] := FALSE;
	garr_stoermeldungen[st_config_achse.i16_meld_startindex + 50] := FALSE;
	garr_stoermeldungen[st_config_achse.i16_meld_startindex + 51] := FALSE;
	garr_stoermeldungen[st_config_achse.i16_meld_startindex + 52] := FALSE;
	garr_stoermeldungen[st_config_achse.i16_meld_startindex + 53] := FALSE;
	garr_stoermeldungen[st_config_achse.i16_meld_startindex + 54] := FALSE;
	garr_stoermeldungen[st_config_achse.i16_meld_startindex + 55] := FALSE;
	garr_stoermeldungen[st_config_achse.i16_meld_startindex + 56] := FALSE;
	garr_stoermeldungen[st_config_achse.i16_meld_startindex + 57] := FALSE;
	garr_stoermeldungen[st_config_achse.i16_meld_startindex + 58] := FALSE;
	garr_stoermeldungen[st_config_achse.i16_meld_startindex + 59] := FALSE;
	garr_stoermeldungen[st_config_achse.i16_meld_startindex + 60] := FALSE;
	garr_stoermeldungen[st_config_achse.i16_meld_startindex + 61] := FALSE;
	garr_stoermeldungen[st_config_achse.i16_meld_startindex + 62] := FALSE;
	garr_stoermeldungen[st_config_achse.i16_meld_startindex + 63] := FALSE;
	garr_stoermeldungen[st_config_achse.i16_meld_startindex + 64] := FALSE;
	garr_stoermeldungen[st_config_achse.i16_meld_startindex + 65] := FALSE;
	garr_stoermeldungen[st_config_achse.i16_meld_startindex + 66] := FALSE;
	garr_stoermeldungen[st_config_achse.i16_meld_startindex + 67] := FALSE;
	garr_stoermeldungen[st_config_achse.i16_meld_startindex + 68] := FALSE;
	garr_stoermeldungen[st_config_achse.i16_meld_startindex + 69] := FALSE;
	garr_stoermeldungen[st_config_achse.i16_meld_startindex + 70] := FALSE;
	garr_stoermeldungen[st_config_achse.i16_meld_startindex + 71] := FALSE;
	garr_stoermeldungen[st_config_achse.i16_meld_startindex + 72] := FALSE;
	garr_stoermeldungen[st_config_achse.i16_meld_startindex + 73] := FALSE;
	garr_stoermeldungen[st_config_achse.i16_meld_startindex + 74] := FALSE;
	garr_stoermeldungen[st_config_achse.i16_meld_startindex + 75] := FALSE;
	garr_stoermeldungen[st_config_achse.i16_meld_startindex + 76] := FALSE;
	garr_stoermeldungen[st_config_achse.i16_meld_startindex + 77] := FALSE;
	garr_stoermeldungen[st_config_achse.i16_meld_startindex + 78] := FALSE;
	garr_stoermeldungen[st_config_achse.i16_meld_startindex + 79] := FALSE;
	garr_stoermeldungen[st_config_achse.i16_meld_startindex + 80] := FALSE;
	garr_stoermeldungen[st_config_achse.i16_meld_startindex + 81] := FALSE;
	garr_stoermeldungen[st_config_achse.i16_meld_startindex + 82] := FALSE;
	garr_stoermeldungen[st_config_achse.i16_meld_startindex + 83] := FALSE;
	garr_stoermeldungen[st_config_achse.i16_meld_startindex + 84] := FALSE;
	garr_stoermeldungen[st_config_achse.i16_meld_startindex + 85] := FALSE;
	garr_stoermeldungen[st_config_achse.i16_meld_startindex + 86] := FALSE;
	garr_stoermeldungen[st_config_achse.i16_meld_startindex + 87] := FALSE;
	garr_stoermeldungen[st_config_achse.i16_meld_startindex + 88] := FALSE;
	garr_stoermeldungen[st_config_achse.i16_meld_startindex + 89] := FALSE;
	garr_stoermeldungen[st_config_achse.i16_meld_startindex + 90] := FALSE;
	garr_stoermeldungen[st_config_achse.i16_meld_startindex + 91] := FALSE;
	garr_stoermeldungen[st_config_achse.i16_meld_startindex + 92] := FALSE;
	garr_stoermeldungen[st_config_achse.i16_meld_startindex + 93] := FALSE;
	garr_stoermeldungen[st_config_achse.i16_meld_startindex + 94] := FALSE;
	garr_stoermeldungen[st_config_achse.i16_meld_startindex + 95] := FALSE;
	garr_stoermeldungen[st_config_achse.i16_meld_startindex + 96] := FALSE;
	garr_stoermeldungen[st_config_achse.i16_meld_startindex + 97] := FALSE;
	garr_stoermeldungen[st_config_achse.i16_meld_startindex + 98] := FALSE;
	garr_stoermeldungen[st_config_achse.i16_meld_startindex + 99] := FALSE;
	
	garr_betriebsmeldungen[st_config_achse.i16_meld_startindex + 0] := FALSE;
	garr_betriebsmeldungen[st_config_achse.i16_meld_startindex + 1] := FALSE;
	garr_betriebsmeldungen[st_config_achse.i16_meld_startindex + 2] := FALSE;
	garr_betriebsmeldungen[st_config_achse.i16_meld_startindex + 3] := FALSE;
	garr_betriebsmeldungen[st_config_achse.i16_meld_startindex + 4] := FALSE;
	garr_betriebsmeldungen[st_config_achse.i16_meld_startindex + 5] := FALSE;
	garr_betriebsmeldungen[st_config_achse.i16_meld_startindex + 6] := FALSE;
	garr_betriebsmeldungen[st_config_achse.i16_meld_startindex + 7] := FALSE;
	garr_betriebsmeldungen[st_config_achse.i16_meld_startindex + 8] := FALSE;
	garr_betriebsmeldungen[st_config_achse.i16_meld_startindex + 9] := FALSE;
	garr_betriebsmeldungen[st_config_achse.i16_meld_startindex + 10] := FALSE;
	garr_betriebsmeldungen[st_config_achse.i16_meld_startindex + 11] := FALSE;
	garr_betriebsmeldungen[st_config_achse.i16_meld_startindex + 12] := FALSE;
	garr_betriebsmeldungen[st_config_achse.i16_meld_startindex + 13] := FALSE;
	garr_betriebsmeldungen[st_config_achse.i16_meld_startindex + 14] := FALSE;
	garr_betriebsmeldungen[st_config_achse.i16_meld_startindex + 15] := FALSE;
	garr_betriebsmeldungen[st_config_achse.i16_meld_startindex + 16] := FALSE;
	garr_betriebsmeldungen[st_config_achse.i16_meld_startindex + 17] := FALSE;
	garr_betriebsmeldungen[st_config_achse.i16_meld_startindex + 18] := FALSE;
	garr_betriebsmeldungen[st_config_achse.i16_meld_startindex + 19] := FALSE;
	garr_betriebsmeldungen[st_config_achse.i16_meld_startindex + 20] := FALSE;
	garr_betriebsmeldungen[st_config_achse.i16_meld_startindex + 21] := FALSE;
	garr_betriebsmeldungen[st_config_achse.i16_meld_startindex + 22] := FALSE;
	garr_betriebsmeldungen[st_config_achse.i16_meld_startindex + 23] := FALSE;
	garr_betriebsmeldungen[st_config_achse.i16_meld_startindex + 24] := FALSE;
	garr_betriebsmeldungen[st_config_achse.i16_meld_startindex + 25] := FALSE;
	garr_betriebsmeldungen[st_config_achse.i16_meld_startindex + 26] := FALSE;
	garr_betriebsmeldungen[st_config_achse.i16_meld_startindex + 27] := FALSE;
	garr_betriebsmeldungen[st_config_achse.i16_meld_startindex + 28] := FALSE;
	garr_betriebsmeldungen[st_config_achse.i16_meld_startindex + 29] := FALSE;
	garr_betriebsmeldungen[st_config_achse.i16_meld_startindex + 30] := FALSE;
	garr_betriebsmeldungen[st_config_achse.i16_meld_startindex + 31] := FALSE;
	garr_betriebsmeldungen[st_config_achse.i16_meld_startindex + 32] := FALSE;
	garr_betriebsmeldungen[st_config_achse.i16_meld_startindex + 33] := FALSE;
	garr_betriebsmeldungen[st_config_achse.i16_meld_startindex + 34] := FALSE;
	garr_betriebsmeldungen[st_config_achse.i16_meld_startindex + 35] := FALSE;
	garr_betriebsmeldungen[st_config_achse.i16_meld_startindex + 36] := FALSE;
	garr_betriebsmeldungen[st_config_achse.i16_meld_startindex + 37] := FALSE;
	garr_betriebsmeldungen[st_config_achse.i16_meld_startindex + 38] := FALSE;
	garr_betriebsmeldungen[st_config_achse.i16_meld_startindex + 39] := FALSE;
	garr_betriebsmeldungen[st_config_achse.i16_meld_startindex + 40] := FALSE;
	garr_betriebsmeldungen[st_config_achse.i16_meld_startindex + 41] := FALSE;
	garr_betriebsmeldungen[st_config_achse.i16_meld_startindex + 42] := FALSE;
	garr_betriebsmeldungen[st_config_achse.i16_meld_startindex + 43] := FALSE;
	garr_betriebsmeldungen[st_config_achse.i16_meld_startindex + 44] := FALSE;
	garr_betriebsmeldungen[st_config_achse.i16_meld_startindex + 45] := FALSE;
	garr_betriebsmeldungen[st_config_achse.i16_meld_startindex + 46] := FALSE;
	garr_betriebsmeldungen[st_config_achse.i16_meld_startindex + 47] := FALSE;
	garr_betriebsmeldungen[st_config_achse.i16_meld_startindex + 48] := FALSE;
	garr_betriebsmeldungen[st_config_achse.i16_meld_startindex + 49] := FALSE;
END_IF
END_PROGRAM
ACTION subr_ST_Vorschubkontrolle:
IF gi16_betriebsart <> HAND AND NOT ST_TippTasten.b_einfaedeln_aktiv AND st_ctrl_in.b_freigabe THEN
(* Warte auf Vorschubnocke  und Freigabe von der Virtuellen Masterachse *)
(* Die Freigabe erfolgt nur im normalen Produktionsablauf; nicht bei Bandwechsel, Einfädeln, ... da hier keine Überwachung erfolgen soll. *)

	(* Am Anfang des Bandvorschubs Zähler zurücksetzen *)
	IF  fb_r_trig_nocke_einzug.Q THEN
		i_zaehler_steigende_flanke := 0;
		i_zaehler_fallende_flanke := 0;
	END_IF

	(* Zähler Vorschubkontrolle durch positive Flanke erhöhen *)
	IF fb_r_trig_vorschubkontrolle.Q THEN
		i_zaehler_steigende_flanke := i_zaehler_steigende_flanke + 1;
	END_IF
	(* Zähler Vorschubkontrolle durch negative Flanke erhöhen *)
	IF fb_f_trig_vorschubkontrolle.Q THEN
		i_zaehler_fallende_flanke := i_zaehler_fallende_flanke + 1;
	END_IF

	(* Am Ende des Bandvorschubs die Zähler mit der Vorgabe vergleichen *)
	IF fb_f_trig_nocke_einzug.Q THEN
		IF 	i_zaehler_steigende_flanke <> gst_datensatz.st_bestueckprogramm.i16_b[ST_Virtuelle_Masterachse.i16_bestueckposzaehler] OR
			i_zaehler_fallende_flanke <> gst_datensatz.st_bestueckprogramm.i16_b[ST_Virtuelle_Masterachse.i16_bestueckposzaehler] THEN
			sm_fehler_bandvorschub := TRUE;
			fb_state_entry.i16_next_step := FEHLER;
		END_IF
	END_IF
ELSE
	i_zaehler_steigende_flanke := 0;
	i_zaehler_fallende_flanke := 0;
END_IF
END_ACTION

(* POU Gemeinsamkeiten17xx/Betriebsarten/ST_Betriebsarten, ST *)
PROGRAM ST_Betriebsarten
VAR_INPUT
	st_config					: struct_config;
END_VAR
VAR
	fb_ton_wz				: TON;
	fb_state_entry				: ST_StateEntry;
	i16_betriebsart 			: enum_betriebsarten := KEINE;
	e_ba_automatik			AT %I* : BOOL;
	e_ba_tippen				AT %I* : BOOL;
	e_ba_hand				AT %I* : BOOL;
	e_ba_dummy				AT %I* : BOOL;
	e_ba_pseudo			AT %I* : BOOL;
	a_lampe_ba_automatik	AT %Q* : BOOL;
	a_lampe_ba_tippen		AT %Q* : BOOL;
	a_lampe_ba_hand		AT %Q* : BOOL;
	a_lampe_ba_dummy		AT %Q* : BOOL;
	a_lampe_ba_pseudo		AT %Q* : BOOL;
END_VAR
gi16_betriebsart := i16_betriebsart;

(* Zeiten *)
fb_ton_wz(IN:= , PT:= t#1s, Q=>  , ET=> );

(* ======================================Schrittkette======================================== *)
fb_state_entry(
	i16_next_step:= ,
	i16_pos:= 1,
	s_debugtext:= ,
	E=> ,
	X=> ,
	i16_step=> ,
	i16_last_step=> );

CASE fb_state_entry.i16_step OF
(*=======================================================*)
	0:	(* KEINE *)
		IF fb_state_entry.E THEN
			fb_ton_wz.IN := TRUE;
		END_IF
		IF fb_ton_wz.Q THEN
			i16_betriebsart := KEINE;
		END_IF

		a_lampe_ba_automatik := FALSE;
		a_lampe_ba_tippen := FALSE;
		a_lampe_ba_hand := FALSE;
		a_lampe_ba_dummy := FALSE;
		a_lampe_ba_pseudo := FALSE;

		(* Betriebsartenwechsel *)
		IF e_ba_automatik THEN
			fb_state_entry.i16_next_step := 10;	(* AUTO *)
		ELSIF e_ba_tippen THEN
			fb_state_entry.i16_next_step := 20;	(* TIPPEN *)
		ELSIF e_ba_hand THEN
			fb_state_entry.i16_next_step := 30;	(* HAND *)
		ELSIF e_ba_dummy THEN
			fb_state_entry.i16_next_step := 40;	(* DUMMY *)
		ELSIF e_ba_pseudo THEN
			fb_state_entry.i16_next_step := 50;	(* PSEUDO *)
		END_IF

(*=======================================================*)
	10:	(* AUTO *)
		IF fb_state_entry.E THEN
			i16_betriebsart := AUTO;
			a_lampe_ba_automatik := TRUE;
		END_IF

		(* Betriebsartenwechsel *)
		IF NOT e_ba_automatik THEN
			fb_state_entry.i16_next_step := 0;
		END_IF
	
	(*=======================================================*)
	20:	(* TIPPEN *)
		IF fb_state_entry.E THEN
			i16_betriebsart := TIPPEN;
			a_lampe_ba_tippen := TRUE;
		END_IF

		(* Betriebsartenwechsel *)
		IF NOT e_ba_tippen THEN
			fb_state_entry.i16_next_step := 0;
		END_IF

(*=======================================================*)
	30:	(* HAND *)
		IF fb_state_entry.E THEN
			i16_betriebsart := HAND;
			a_lampe_ba_hand := TRUE;
		END_IF

		(* Betriebsartenwechsel *)
		IF NOT e_ba_hand THEN
			fb_state_entry.i16_next_step := 0;
		END_IF

(*=======================================================*)
	40:	(* DUMMY *)
		IF fb_state_entry.E THEN
			i16_betriebsart := DUMMY;
			a_lampe_ba_dummy := TRUE;
		END_IF

		(* Betriebsartenwechsel *)
		IF NOT e_ba_dummy THEN
			fb_state_entry.i16_next_step := 0;
		END_IF

(*=======================================================*)
	50:	(* PSEUDO *)
		IF fb_state_entry.E THEN
			i16_betriebsart := PSEUDO;
			a_lampe_ba_pseudo := TRUE;
		END_IF

		(* Betriebsartenwechsel *)
		IF NOT e_ba_pseudo THEN
			fb_state_entry.i16_next_step := 0;
		END_IF
END_CASE

fb_state_entry(
	i16_next_step:= ,
	i16_pos:= 2,
	s_debugtext:= ,
	E=> , 
	X=> , 
	i16_step=> ,
	i16_last_step=> );

IF st_config.b_config_fertig THEN
	(* Fehlermeldungen  *)
	garr_stoermeldungen[st_config.i16_meld_startindex + 0] := FALSE;
	garr_stoermeldungen[st_config.i16_meld_startindex + 1] := FALSE;
	garr_stoermeldungen[st_config.i16_meld_startindex + 2] := FALSE;
	garr_stoermeldungen[st_config.i16_meld_startindex + 3] := FALSE;
	garr_stoermeldungen[st_config.i16_meld_startindex + 4] := FALSE;
	garr_stoermeldungen[st_config.i16_meld_startindex + 5] := FALSE;
	garr_stoermeldungen[st_config.i16_meld_startindex + 6] := FALSE;
	garr_stoermeldungen[st_config.i16_meld_startindex + 7] := FALSE;
	garr_stoermeldungen[st_config.i16_meld_startindex + 8] := FALSE;
	garr_stoermeldungen[st_config.i16_meld_startindex + 9] := FALSE;
	garr_stoermeldungen[st_config.i16_meld_startindex + 10] := FALSE;
	garr_stoermeldungen[st_config.i16_meld_startindex + 11] := FALSE;
	garr_stoermeldungen[st_config.i16_meld_startindex + 12] := FALSE;
	garr_stoermeldungen[st_config.i16_meld_startindex + 13] := FALSE;
	garr_stoermeldungen[st_config.i16_meld_startindex + 14] := FALSE;
	garr_stoermeldungen[st_config.i16_meld_startindex + 15] := FALSE;
	garr_stoermeldungen[st_config.i16_meld_startindex + 16] := FALSE;
	garr_stoermeldungen[st_config.i16_meld_startindex + 17] := FALSE;
	garr_stoermeldungen[st_config.i16_meld_startindex + 18] := FALSE;
	garr_stoermeldungen[st_config.i16_meld_startindex + 19] := FALSE;
	
	(* Betriebsmeldungen *)
	garr_betriebsmeldungen[st_config.i16_meld_startindex + 0] := FALSE;
	garr_betriebsmeldungen[st_config.i16_meld_startindex + 1] := FALSE;
	garr_betriebsmeldungen[st_config.i16_meld_startindex + 2] := FALSE;
	garr_betriebsmeldungen[st_config.i16_meld_startindex + 3] := FALSE;
	garr_betriebsmeldungen[st_config.i16_meld_startindex + 4] := FALSE;
	garr_betriebsmeldungen[st_config.i16_meld_startindex + 5] := FALSE;
	garr_betriebsmeldungen[st_config.i16_meld_startindex + 6] := FALSE;
	garr_betriebsmeldungen[st_config.i16_meld_startindex + 7] := FALSE;
	garr_betriebsmeldungen[st_config.i16_meld_startindex + 8] := FALSE;
	garr_betriebsmeldungen[st_config.i16_meld_startindex + 9] := FALSE;
	garr_betriebsmeldungen[st_config.i16_meld_startindex + 10] := FALSE;
	garr_betriebsmeldungen[st_config.i16_meld_startindex + 11] := FALSE;
	garr_betriebsmeldungen[st_config.i16_meld_startindex + 12] := FALSE;
	garr_betriebsmeldungen[st_config.i16_meld_startindex + 13] := FALSE;
	garr_betriebsmeldungen[st_config.i16_meld_startindex + 14] := FALSE;
	garr_betriebsmeldungen[st_config.i16_meld_startindex + 15] := FALSE;
	garr_betriebsmeldungen[st_config.i16_meld_startindex + 16] := FALSE;
	garr_betriebsmeldungen[st_config.i16_meld_startindex + 17] := FALSE;
	garr_betriebsmeldungen[st_config.i16_meld_startindex + 18] := FALSE;
	garr_betriebsmeldungen[st_config.i16_meld_startindex + 19] := FALSE;
END_IF
END_PROGRAM

(* POU Gemeinsamkeiten17xx/Achsen/F_Servobandeinzug_Strecke_zu_Grad, ST *)
FUNCTION F_Servobandeinzug_Strecke_zu_Grad : LREAL
VAR_INPUT
	strecke	: LREAL;
END_VAR
VAR
	Umfang : LREAL;
END_VAR
Umfang :=  gst_datensatz.st_band.i16_igelrad_zaehne * gst_datensatz.st_band.r_raster;
lr_debug :=  (360.0 * strecke ) / Umfang ;
F_Servobandeinzug_Strecke_zu_Grad := lr_debug;
END_FUNCTION

(* POU Gemeinsamkeiten17xx/Achsen/F_Startpos_Servobandeinzug, ST *)
FUNCTION F_Startpos_Servobandeinzug : LREAL
VAR_INPUT
	r_actual_pos : LREAL:= 1.0;
END_VAR
VAR
	i16_gerundet : INT:= 0;
	startpos : INT := 3;
	i16_grad_pro_zahn : INT := 10;
	r_grad_pro_zahn : LREAL := 10.0;
END_VAR
(* Das Igelrad muss zum Einfädeln an einer bestimmten Gradzahl stehen.
Diese ist abhängig von der größe des Igelrads *)

i16_gerundet := LREAL_TO_INT(r_actual_pos/r_grad_pro_zahn);

F_Startpos_Servobandeinzug := INT_TO_LREAL(i16_gerundet * i16_grad_pro_zahn - gst_datensatz.st_band.i16_startpos_einfaedeln);
END_FUNCTION

(* POU Gemeinsamkeiten17xx/TagReader/ST_Markiere_WT_NIO, ST *)
PROGRAM ST_Markiere_WT_NIO
VAR
	i : INT := 0;
END_VAR
IF gst_datensatz.st_md.i16_tag_data_structur_version = 0 THEN
	gst_tag_data.StateParts[0] := PART_NOK;
	gst_tag_data.StateParts[1] := PART_NOK;

	(* Starte Schreib Prozess *)
	balluff_tag_reader.fb.i16_addresse := 1;
	balluff_tag_reader.fb.i16_anzahl_byte := 2;
	balluff_tag_reader.fb.s_schreib_daten[0] := DINT_TO_BYTE(gst_tag_data.StateParts[0]);
	balluff_tag_reader.fb.s_schreib_daten[1] := DINT_TO_BYTE(gst_tag_data.StateParts[1]);
	balluff_tag_reader.st_ctrl.in.b_start_schreiben := TRUE;
ELSIF gst_datensatz.st_md.i16_tag_data_structur_version = 1 THEN
	balluff_tag_reader.fb.i16_addresse := 1;
	balluff_tag_reader.fb.i16_anzahl_byte := 8;
	FOR i:= 0 TO gst_tag_data.AmountPartsOnWpc - 1 BY 1 DO
		gst_tag_data.StateParts[i] := PART_NOK;
	END_FOR
	FOR i:= gst_tag_data.AmountPartsOnWpc TO 7 BY 1 DO
		gst_tag_data.StateParts[i] := PART_NO;
	END_FOR
	FOR i:= 0 TO 7 BY 1 DO
		balluff_tag_reader.fb.s_schreib_daten[i] := DINT_TO_BYTE(gst_tag_data.StateParts[i]);
	END_FOR
	balluff_tag_reader.st_ctrl.in.b_start_schreiben := TRUE;
END_IF
END_PROGRAM

(* POU Gemeinsamkeiten17xx/TagReader/ST_Markiere_WT_IO, ST *)
PROGRAM ST_Markiere_WT_IO
VAR
	i 						:INT := 0;
	b_Rasterfolie_montiert	:BOOL;
END_VAR
(* Auswertung der Bestückung (Pins bzw. Rasterplatte) des ISK *)
CASE gst_datensatz.st_md.i16_typ_zelle OF
	KEINE_ZELLE:
		;

